LIN {X 0,Y 313.561,Z 316.467,A -85,B 0,C 180,E1 -15772.474,E2 -15772.474} C_VEL
LIN {X 0,Y 320.845,Z 338.006,A -85,B 0,C 180,E1 -15773.542,E2 -15773.542} C_VEL
LIN {X 0,Y 322.386,Z 346.746,A -85,B 0,C 180,E1 -15773.871,E2 -15773.871} C_VEL
LIN {X 0,Y 320.224,Z 424.19,A -85,B 0,C 180,E1 -15775.8,E2 -15775.8} C_VEL
LIN {X 0,Y 319.459,Z 438.164,A -85,B 0,C 180,E1 -15776.412,E2 -15776.412} C_VEL
LIN {X 0,Y 318.685,Z 450.762,A -85,B 0,C 180,E1 -15777.233,E2 -15777.233} C_VEL
LIN {X 0,Y 317.606,Z 462.924,A -85,B 0,C 180,E1 -15778.297,E2 -15778.297} C_VEL
LIN {X 0,Y 316.488,Z 474.165,A -85,B 0,C 180,E1 -15779.558,E2 -15779.558} C_VEL
LIN {X 0,Y 315.388,Z 484.512,A -85,B 0,C 180,E1 -15781.019,E2 -15781.019} C_VEL
LIN {X 0,Y 314.251,Z 493.873,A -85,B 0,C 180,E1 -15782.653,E2 -15782.653} C_VEL
LIN {X 0,Y 313.15,Z 502.541,A -85,B 0,C 180,E1 -15784.52,E2 -15784.52} C_VEL
LIN {X 0,Y 312.337,Z 509.035,A -85,B 0,C 180,E1 -15786.251,E2 -15786.251} C_VEL
LIN {X 0,Y 311.635,Z 515.662,A -85,B 0,C 180,E1 -15788.494,E2 -15788.494} C_VEL
LIN {X 0,Y 311.223,Z 519.919,A -85,B 0,C 180,E1 -15790.35,E2 -15790.35} C_VEL
LIN {X 0,Y 310.751,Z 523.922,A -85,B 0,C 180,E1 -15792.726,E2 -15792.726} C_VEL
LIN {X 0,Y 310.539,Z 525.963,A -85,B 0,C 180,E1 -15794.555,E2 -15794.555} C_VEL
LIN {X 0,Y 310.509,Z 527.474,A -85,B 0,C 180,E1 -15797.233,E2 -15797.233} C_VEL
LIN {X 0,Y 310.562,Z 527.524,A -85,B 0,C 180,E1 -15798.983,E2 -15798.983} C_VEL
LIN {X 0,Y 310.752,Z 526.817,A -85,B 0,C 180,E1 -15800.709,E2 -15800.709} C_VEL
LIN {X 0,Y 311.274,Z 524.504,A -85,B 0,C 180,E1 -15803.25,E2 -15803.25} C_VEL
LIN {X 0,Y 311.79,Z 521.895,A -85,B 0,C 180,E1 -15805.018,E2 -15805.018} C_VEL
LIN {X 0,Y 312.69,Z 517.119,A -85,B 0,C 180,E1 -15807.355,E2 -15807.355} C_VEL
LIN {X 0,Y 313.24,Z 514.23,A -85,B 0,C 180,E1 -15808.473,E2 -15808.473} C_VEL
LIN {X 0,Y 313.144,Z 511.578,A -85,B 0,C 180,E1 -15809.439,E2 -15809.439} C_VEL
LIN {X 0,Y 311.349,Z 506.988,A -85,B 0,C 180,E1 -15811.019,E2 -15811.019} C_VEL
LIN {X 0,Y 309.655,Z 501.778,A -85,B 0,C 180,E1 -15812.544,E2 -15812.544} C_VEL
LIN {X 0,Y 309.708,Z 498.155,A -85,B 0,C 180,E1 -15813.407,E2 -15813.407} C_VEL
LIN {X 0,Y 311.191,Z 489.974,A -85,B 0,C 180,E1 -15815.021,E2 -15815.021} C_VEL
LIN {X 0,Y 312.898,Z 480.264,A -85,B 0,C 180,E1 -15816.569,E2 -15816.569} C_VEL
LIN {X 0,Y 314.489,Z 470.173,A -85,B 0,C 180,E1 -15817.862,E2 -15817.862} C_VEL
LIN {X 0,Y 316.068,Z 458.486,A -85,B 0,C 180,E1 -15819.052,E2 -15819.052} C_VEL
LIN {X 0,Y 317.448,Z 446.076,A -85,B 0,C 180,E1 -15820.015,E2 -15820.015} C_VEL
LIN {X 0,Y 318.404,Z 433.369,A -85,B 0,C 180,E1 -15820.729,E2 -15820.729} C_VEL
LIN {X 0,Y 319.199,Z 419.555,A -85,B 0,C 180,E1 -15821.22,E2 -15821.22} C_VEL
LIN {X 0,Y 321.928,Z 348.78,A -85,B 0,C 180,E1 -15823.058,E2 -15823.058} C_VEL
LIN {X 0,Y 315.974,Z 334.725,A -85,B 0,C 180,E1 -15824.194,E2 -15824.194} C_VEL
LIN {X 0,Y 308.836,Z 320.932,A -85,B 0,C 180,E1 -15825.566,E2 -15825.566} C_VEL
LIN {X 0,Y 307.107,Z 317.583,A -85,B 0,C 180,E1 -15825.927,E2 -15825.927} C_VEL
LIN {X 0,Y 305.593,Z 312.421,A -85,B 0,C 180,E1 -15827.717,E2 -15827.717} C_VEL
LIN {X 0,Y 305.815,Z 312.391,A -85,B 0,C 180,E1 -15832.074,E2 -15832.074} C_VEL
LIN {X 0,Y 305.69,Z 312.409,A -85,B 0,C 180,E1 -15834.723,E2 -15834.723} C_VEL
LIN {X 0,Y 305.958,Z 312.371,A -85,B 0,C 180,E1 -15838.683,E2 -15838.683} C_VEL
LIN {X 0,Y 305.958,Z 312.368,A -85,B 0,C 180,E1 -15841.316,E2 -15841.316} C_VEL
LIN {X 0,Y 305.678,Z 312.408,A -85,B 0,C 180,E1 -15845.276,E2 -15845.276} C_VEL
LIN {X 0,Y 305.767,Z 312.393,A -85,B 0,C 180,E1 -15847.927,E2 -15847.927} C_VEL
LIN {X 0,Y 305.606,Z 312.418,A -85,B 0,C 180,E1 -15851.945,E2 -15851.945} C_VEL
LIN {X 0,Y 305.612,Z 312.417,A -85,B 0,C 180,E1 -15855.015,E2 -15855.015} C_VEL
LIN {X 0,Y 305.544,Z 312.424,A -85,B 0,C 180,E1 -15859.426,E2 -15859.426} C_VEL
LIN {X 0,Y 305.488,Z 312.43,A -85,B 0,C 180,E1 -15863.039,E2 -15863.039} C_VEL
LIN {X 0,Y 305.549,Z 312.423,A -85,B 0,C 180,E1 -15866.226,E2 -15866.226} C_VEL
LIN {X 0,Y 305.49,Z 312.427,A -85,B 0,C 180,E1 -15869.047,E2 -15869.047} C_VEL
LIN {X 0,Y 305.444,Z 312.431,A -85,B 0,C 180,E1 -15871.952,E2 -15871.952} C_VEL
LIN {X 0,Y 305.464,Z 312.43,A -85,B 0,C 180,E1 -15875.113,E2 -15875.113} C_VEL
LIN {X 0,Y 305.442,Z 312.434,A -85,B 0,C 180,E1 -15878.526,E2 -15878.526} C_VEL
LIN {X 0,Y 305.457,Z 312.438,A -85,B 0,C 180,E1 -15882.585,E2 -15882.585} C_VEL
LIN {X 0,Y 305.427,Z 312.438,A -85,B 0,C 180,E1 -15886.345,E2 -15886.345} C_VEL
LIN {X 0,Y 305.46,Z 312.434,A -85,B 0,C 180,E1 -15889.892,E2 -15889.892} C_VEL
LIN {X 0,Y 305.509,Z 312.492,A -85,B 0,C 180,E1 -15894.134,E2 -15894.134} C_VEL
LIN {X 0,Y 308.452,Z 323.369,A -85,B 0,C 180,E1 -15897.885,E2 -15897.885} C_VEL
LIN {X 0,Y 310.938,Z 334.197,A -85,B 0,C 180,E1 -15901.294,E2 -15901.294} C_VEL
LIN {X 0,Y 311.28,Z 335.799,A -85,B 0,C 180,E1 -15901.707,E2 -15901.707} C_VEL
LIN {X 0,Y 314.458,Z 343.704,A -85,B 0,C 180,E1 -15902.366,E2 -15902.366} C_VEL
LIN {X 0,Y 318.425,Z 363.354,A -85,B 0,C 180,E1 -15903.452,E2 -15903.452} C_VEL
LIN {X 0,Y 320.87,Z 381.215,A -85,B 0,C 180,E1 -15904.276,E2 -15904.276} C_VEL
LIN {X 0,Y 318.482,Z 445.12,A -85,B 0,C 180,E1 -15905.948,E2 -15905.948} C_VEL
LIN {X 0,Y 317.369,Z 459.165,A -85,B 0,C 180,E1 -15906.552,E2 -15906.552} C_VEL
LIN {X 0,Y 315.998,Z 471.837,A -85,B 0,C 180,E1 -15907.353,E2 -15907.353} C_VEL
LIN {X 0,Y 314.357,Z 483.549,A -85,B 0,C 180,E1 -15908.352,E2 -15908.352} C_VEL
LIN {X 0,Y 312.61,Z 494.909,A -85,B 0,C 180,E1 -15909.606,E2 -15909.606} C_VEL
LIN {X 0,Y 310.852,Z 505.242,A -85,B 0,C 180,E1 -15911.034,E2 -15911.034} C_VEL
LIN {X 0,Y 309.342,Z 513.737,A -85,B 0,C 180,E1 -15912.48,E2 -15912.48} C_VEL
LIN {X 0,Y 307.656,Z 523.012,A -85,B 0,C 180,E1 -15914.429,E2 -15914.429} C_VEL
LIN {X 0,Y 306.221,Z 530.528,A -85,B 0,C 180,E1 -15916.393,E2 -15916.393} C_VEL
LIN {X 0,Y 305.201,Z 535.652,A -85,B 0,C 180,E1 -15918.038,E2 -15918.038} C_VEL
LIN {X 0,Y 304.451,Z 540.647,A -85,B 0,C 180,E1 -15920.029,E2 -15920.029} C_VEL
LIN {X 0,Y 303.956,Z 544.511,A -85,B 0,C 180,E1 -15922.025,E2 -15922.025} C_VEL
LIN {X 0,Y 303.625,Z 547.846,A -85,B 0,C 180,E1 -15924.455,E2 -15924.455} C_VEL
LIN {X 0,Y 303.631,Z 549.216,A -85,B 0,C 180,E1 -15926.017,E2 -15926.017} C_VEL
LIN {X 0,Y 303.623,Z 549.939,A -85,B 0,C 180,E1 -15927.346,E2 -15927.346} C_VEL
LIN {X 0,Y 303.613,Z 550.264,A -85,B 0,C 180,E1 -15928.673,E2 -15928.673} C_VEL
LIN {X 0,Y 303.669,Z 550.168,A -85,B 0,C 180,E1 -15929.999,E2 -15929.999} C_VEL
LIN {X 0,Y 303.626,Z 549.623,A -85,B 0,C 180,E1 -15931.326,E2 -15931.326} C_VEL
LIN {X 0,Y 303.63,Z 548.674,A -85,B 0,C 180,E1 -15932.653,E2 -15932.653} C_VEL
LIN {X 0,Y 303.655,Z 547.312,A -85,B 0,C 180,E1 -15933.981,E2 -15933.981} C_VEL
LIN {X 0,Y 303.665,Z 544.964,A -85,B 0,C 180,E1 -15935.621,E2 -15935.621} C_VEL
LIN {X 0,Y 303.939,Z 540.379,A -85,B 0,C 180,E1 -15937.974,E2 -15937.974} C_VEL
LIN {X 0,Y 304.443,Z 534.159,A -85,B 0,C 180,E1 -15940.305,E2 -15940.305} C_VEL
LIN {X 0,Y 305.146,Z 527.327,A -85,B 0,C 180,E1 -15942.3,E2 -15942.3} C_VEL
LIN {X 0,Y 306.186,Z 518.829,A -85,B 0,C 180,E1 -15944.284,E2 -15944.284} C_VEL
LIN {X 0,Y 307.231,Z 510.041,A -85,B 0,C 180,E1 -15945.932,E2 -15945.932} C_VEL
LIN {X 0,Y 308.372,Z 500.41,A -85,B 0,C 180,E1 -15947.404,E2 -15947.404} C_VEL
LIN {X 0,Y 309.563,Z 489.924,A -85,B 0,C 180,E1 -15948.703,E2 -15948.703} C_VEL
LIN {X 0,Y 310.837,Z 478.475,A -85,B 0,C 180,E1 -15949.824,E2 -15949.824} C_VEL
LIN {X 0,Y 312.023,Z 465.463,A -85,B 0,C 180,E1 -15950.777,E2 -15950.777} C_VEL
LIN {X 0,Y 312.903,Z 452.597,A -85,B 0,C 180,E1 -15951.449,E2 -15951.449} C_VEL
LIN {X 0,Y 313.47,Z 439.226,A -85,B 0,C 180,E1 -15951.883,E2 -15951.883} C_VEL
LIN {X 0,Y 314.956,Z 378.874,A -85,B 0,C 180,E1 -15953.412,E2 -15953.412} C_VEL
LIN {X 0,Y 309.275,Z 338.42,A -85,B 0,C 180,E1 -15954.905,E2 -15954.905} C_VEL
LIN {X 0,Y 309.725,Z 333.405,A -85,B 0,C 180,E1 -15956.261,E2 -15956.261} C_VEL
LIN {X 0,Y 307.875,Z 323.557,A -85,B 0,C 180,E1 -15959.147,E2 -15959.147} C_VEL
LIN {X 0,Y 305.484,Z 312.437,A -85,B 0,C 180,E1 -15962.58,E2 -15962.58} C_VEL
LIN {X 0,Y 305.472,Z 312.434,A -85,B 0,C 180,E1 -15966.739,E2 -15966.739} C_VEL
LIN {X 0,Y 305.451,Z 312.437,A -85,B 0,C 180,E1 -15970.599,E2 -15970.599} C_VEL
LIN {X 0,Y 305.422,Z 312.437,A -85,B 0,C 180,E1 -15973.654,E2 -15973.654} C_VEL
LIN {X 0,Y 305.451,Z 312.434,A -85,B 0,C 180,E1 -15977.413,E2 -15977.413} C_VEL
LIN {X 0,Y 305.491,Z 312.429,A -85,B 0,C 180,E1 -15981.6,E2 -15981.6} C_VEL
LIN {X 0,Y 305.458,Z 312.437,A -85,B 0,C 180,E1 -15984.886,E2 -15984.886} C_VEL
LIN {X 0,Y 305.444,Z 312.434,A -85,B 0,C 180,E1 -15988.355,E2 -15988.355} C_VEL
LIN {X 0,Y 305.508,Z 312.429,A -85,B 0,C 180,E1 -15991.113,E2 -15991.113} C_VEL
LIN {X 0,Y 305.56,Z 312.42,A -85,B 0,C 180,E1 -15994.087,E2 -15994.087} C_VEL
LIN {X 0,Y 305.495,Z 312.428,A -85,B 0,C 180,E1 -15998.403,E2 -15998.403} C_VEL
LIN {X 0,Y 305.585,Z 312.422,A -85,B 0,C 180,E1 -16001.218,E2 -16001.218} C_VEL
LIN {X 0,Y 305.644,Z 312.414,A -85,B 0,C 180,E1 -16005.349,E2 -16005.349} C_VEL
LIN {X 0,Y 305.633,Z 312.415,A -85,B 0,C 180,E1 -16009.4,E2 -16009.4} C_VEL
LIN {X 0,Y 305.807,Z 312.39,A -85,B 0,C 180,E1 -16012.074,E2 -16012.074} C_VEL
LIN {X 0,Y 305.683,Z 312.404,A -85,B 0,C 180,E1 -16014.724,E2 -16014.724} C_VEL
LIN {X 0,Y 305.951,Z 312.368,A -85,B 0,C 180,E1 -16018.684,E2 -16018.684} C_VEL
LIN {X 0,Y 305.95,Z 312.371,A -85,B 0,C 180,E1 -16021.317,E2 -16021.317} C_VEL
LIN {X 0,Y 305.671,Z 312.406,A -85,B 0,C 180,E1 -16025.277,E2 -16025.277} C_VEL
LIN {X 0,Y 305.76,Z 312.399,A -85,B 0,C 180,E1 -16027.927,E2 -16027.927} C_VEL
LIN {X 0,Y 305.598,Z 312.417,A -85,B 0,C 180,E1 -16031.946,E2 -16031.946} C_VEL
LIN {X 0,Y 305.633,Z 312.409,A -85,B 0,C 180,E1 -16035.035,E2 -16035.035} C_VEL
LIN {X 0,Y 305.575,Z 312.419,A -85,B 0,C 180,E1 -16038.784,E2 -16038.784} C_VEL
LIN {X 0,Y 305.482,Z 312.428,A -85,B 0,C 180,E1 -16043.04,E2 -16043.04} C_VEL
LIN {X 0,Y 305.466,Z 312.431,A -85,B 0,C 180,E1 -16046.198,E2 -16046.198} C_VEL
LIN {X 0,Y 305.454,Z 312.433,A -85,B 0,C 180,E1 -16049.038,E2 -16049.038} C_VEL
LIN {X 0,Y 305.433,Z 312.436,A -85,B 0,C 180,E1 -16051.954,E2 -16051.954} C_VEL
LIN {X 0,Y 305.459,Z 312.434,A -85,B 0,C 180,E1 -16055.114,E2 -16055.114} C_VEL
LIN {X 0,Y 305.432,Z 312.438,A -85,B 0,C 180,E1 -16058.526,E2 -16058.526} C_VEL
LIN {X 0,Y 305.437,Z 312.433,A -85,B 0,C 180,E1 -16061.858,E2 -16061.858} C_VEL
LIN {X 0,Y 305.398,Z 312.441,A -85,B 0,C 180,E1 -16065.512,E2 -16065.512} C_VEL
LIN {X 0,Y 305.41,Z 312.438,A -85,B 0,C 180,E1 -16068.139,E2 -16068.139} C_VEL
LIN {X 0,Y 305.459,Z 312.432,A -85,B 0,C 180,E1 -16071.596,E2 -16071.596} C_VEL
LIN {X 0,Y 305.462,Z 312.433,A -85,B 0,C 180,E1 -16074.888,E2 -16074.888} C_VEL
LIN {X 0,Y 305.442,Z 312.434,A -85,B 0,C 180,E1 -16078.359,E2 -16078.359} C_VEL
LIN {X 0,Y 305.475,Z 312.433,A -85,B 0,C 180,E1 -16081.11,E2 -16081.11} C_VEL
LIN {X 0,Y 305.499,Z 312.428,A -85,B 0,C 180,E1 -16084.082,E2 -16084.082} C_VEL
LIN {X 0,Y 305.475,Z 312.43,A -85,B 0,C 180,E1 -16088.402,E2 -16088.402} C_VEL
LIN {X 0,Y 305.545,Z 312.423,A -85,B 0,C 180,E1 -16091.216,E2 -16091.216} C_VEL
LIN {X 0,Y 305.63,Z 312.413,A -85,B 0,C 180,E1 -16095.349,E2 -16095.349} C_VEL
LIN {X 0,Y 305.626,Z 312.413,A -85,B 0,C 180,E1 -16099.4,E2 -16099.4} C_VEL
LIN {X 0,Y 305.749,Z 312.401,A -85,B 0,C 180,E1 -16102.074,E2 -16102.074} C_VEL
LIN {X 0,Y 305.656,Z 312.409,A -85,B 0,C 180,E1 -16104.724,E2 -16104.724} C_VEL
LIN {X 0,Y 305.934,Z 312.375,A -85,B 0,C 180,E1 -16108.684,E2 -16108.684} C_VEL
LIN {X 0,Y 305.934,Z 312.374,A -85,B 0,C 180,E1 -16111.317,E2 -16111.317} C_VEL
LIN {X 0,Y 305.789,Z 312.395,A -85,B 0,C 180,E1 -16116.599,E2 -16116.599} C_VEL
LIN {X 0,Y 305.687,Z 312.404,A -85,B 0,C 180,E1 -16119.262,E2 -16119.262} C_VEL
LIN {X 0,Y 305.557,Z 312.421,A -85,B 0,C 180,E1 -16123.298,E2 -16123.298} C_VEL
LIN {X 0,Y 305.5,Z 312.429,A -85,B 0,C 180,E1 -16126.026,E2 -16126.026} C_VEL
LIN {X 0,Y 305.507,Z 312.43,A -85,B 0,C 180,E1 -16130.186,E2 -16130.186} C_VEL
LIN {X 0,Y 305.539,Z 312.645,A -85,B 0,C 180,E1 -16130.624,E2 -16130.624} C_VEL
LIN {X 0,Y 306.386,Z 316.706,A -85,B 0,C 180,E1 -16131.974,E2 -16131.974} C_VEL
LIN {X 0,Y 314.265,Z 339.597,A -85,B 0,C 180,E1 -16133.157,E2 -16133.157} C_VEL
LIN {X 0,Y 315.68,Z 347.88,A -85,B 0,C 180,E1 -16133.474,E2 -16133.474} C_VEL
LIN {X 0,Y 313.45,Z 424.389,A -85,B 0,C 180,E1 -16135.424,E2 -16135.424} C_VEL
LIN {X 0,Y 312.68,Z 438.133,A -85,B 0,C 180,E1 -16136.036,E2 -16136.036} C_VEL
LIN {X 0,Y 311.857,Z 450.91,A -85,B 0,C 180,E1 -16136.881,E2 -16136.881} C_VEL
LIN {X 0,Y 310.757,Z 463.159,A -85,B 0,C 180,E1 -16137.975,E2 -16137.975} C_VEL
LIN {X 0,Y 309.631,Z 473.993,A -85,B 0,C 180,E1 -16139.21,E2 -16139.21} C_VEL
LIN {X 0,Y 308.502,Z 484.193,A -85,B 0,C 180,E1 -16140.66,E2 -16140.66} C_VEL
LIN {X 0,Y 307.265,Z 494.192,A -85,B 0,C 180,E1 -16142.437,E2 -16142.437} C_VEL
LIN {X 0,Y 306.173,Z 502.547,A -85,B 0,C 180,E1 -16144.273,E2 -16144.273} C_VEL
LIN {X 0,Y 305.23,Z 509.94,A -85,B 0,C 180,E1 -16146.303,E2 -16146.303} C_VEL
LIN {X 0,Y 304.539,Z 516.295,A -85,B 0,C 180,E1 -16148.543,E2 -16148.543} C_VEL
LIN {X 0,Y 304.131,Z 520.235,A -85,B 0,C 180,E1 -16150.319,E2 -16150.319} C_VEL
LIN {X 0,Y 303.752,Z 523.501,A -85,B 0,C 180,E1 -16152.234,E2 -16152.234} C_VEL
LIN {X 0,Y 303.487,Z 525.806,A -85,B 0,C 180,E1 -16154.119,E2 -16154.119} C_VEL
LIN {X 0,Y 303.406,Z 527.229,A -85,B 0,C 180,E1 -16155.979,E2 -16155.979} C_VEL
LIN {X 0,Y 303.434,Z 527.824,A -85,B 0,C 180,E1 -16157.832,E2 -16157.832} C_VEL
LIN {X 0,Y 303.537,Z 527.598,A -85,B 0,C 180,E1 -16159.825,E2 -16159.825} C_VEL
LIN {X 0,Y 303.865,Z 526.429,A -85,B 0,C 180,E1 -16161.849,E2 -16161.849} C_VEL
LIN {X 0,Y 304.367,Z 524.234,A -85,B 0,C 180,E1 -16163.918,E2 -16163.918} C_VEL
LIN {X 0,Y 305.079,Z 520.889,A -85,B 0,C 180,E1 -16166.03,E2 -16166.03} C_VEL
LIN {X 0,Y 306.023,Z 516.223,A -85,B 0,C 180,E1 -16168.183,E2 -16168.183} C_VEL
LIN {X 0,Y 307.293,Z 510.044,A -85,B 0,C 180,E1 -16170.353,E2 -16170.353} C_VEL
LIN {X 0,Y 308.954,Z 502.039,A -85,B 0,C 180,E1 -16172.519,E2 -16172.519} C_VEL
LIN {X 0,Y 309.708,Z 498.155,A -85,B 0,C 180,E1 -16173.407,E2 -16173.407} C_VEL
LIN {X 0,Y 309.803,Z 494.364,A -85,B 0,C 180,E1 -16174.248,E2 -16174.248} C_VEL
LIN {X 0,Y 308.349,Z 488.096,A -85,B 0,C 180,E1 -16175.651,E2 -16175.651} C_VEL
LIN {X 0,Y 306.955,Z 481.314,A -85,B 0,C 180,E1 -16176.965,E2 -16176.965} C_VEL
LIN {X 0,Y 307.114,Z 476.728,A -85,B 0,C 180,E1 -16177.654,E2 -16177.654} C_VEL
LIN {X 0,Y 308.772,Z 465.962,A -85,B 0,C 180,E1 -16178.941,E2 -16178.941} C_VEL
LIN {X 0,Y 310.429,Z 453.911,A -85,B 0,C 180,E1 -16180.062,E2 -16180.062} C_VEL
LIN {X 0,Y 311.678,Z 441.042,A -85,B 0,C 180,E1 -16180.973,E2 -16180.973} C_VEL
LIN {X 0,Y 312.603,Z 428.721,A -85,B 0,C 180,E1 -16181.571,E2 -16181.571} C_VEL
LIN {X 0,Y 313.553,Z 407.426,A -85,B 0,C 180,E1 -16182.195,E2 -16182.195} C_VEL
LIN {X 0,Y 315.883,Z 351.291,A -85,B 0,C 180,E1 -16183.681,E2 -16183.681} C_VEL
LIN {X 0,Y 314.794,Z 347.909,A -85,B 0,C 180,E1 -16183.918,E2 -16183.918} C_VEL
LIN {X 0,Y 309.105,Z 335.149,A -85,B 0,C 180,E1 -16185.053,E2 -16185.053} C_VEL
LIN {X 0,Y 301.911,Z 321.533,A -85,B 0,C 180,E1 -16186.517,E2 -16186.517} C_VEL
LIN {X 0,Y 299.925,Z 317.942,A -85,B 0,C 180,E1 -16186.965,E2 -16186.965} C_VEL
LIN {X 0,Y 298.568,Z 313.295,A -85,B 0,C 180,E1 -16188.716,E2 -16188.716} C_VEL
LIN {X 0,Y 298.759,Z 313.27,A -85,B 0,C 180,E1 -16191.886,E2 -16191.886} C_VEL
LIN {X 0,Y 298.661,Z 313.285,A -85,B 0,C 180,E1 -16194.599,E2 -16194.599} C_VEL
LIN {X 0,Y 298.924,Z 313.246,A -85,B 0,C 180,E1 -16198.652,E2 -16198.652} C_VEL
LIN {X 0,Y 298.924,Z 313.244,A -85,B 0,C 180,E1 -16201.347,E2 -16201.347} C_VEL
LIN {X 0,Y 298.646,Z 313.284,A -85,B 0,C 180,E1 -16205.401,E2 -16205.401} C_VEL
LIN {X 0,Y 298.715,Z 313.273,A -85,B 0,C 180,E1 -16208.115,E2 -16208.115} C_VEL
LIN {X 0,Y 298.555,Z 313.296,A -85,B 0,C 180,E1 -16212.231,E2 -16212.231} C_VEL
LIN {X 0,Y 298.552,Z 313.296,A -85,B 0,C 180,E1 -16215.169,E2 -16215.169} C_VEL
LIN {X 0,Y 298.505,Z 313.301,A -85,B 0,C 180,E1 -16219.245,E2 -16219.245} C_VEL
LIN {X 0,Y 298.431,Z 313.307,A -85,B 0,C 180,E1 -16223.6,E2 -16223.6} C_VEL
LIN {X 0,Y 298.491,Z 313.303,A -85,B 0,C 180,E1 -16226.574,E2 -16226.574} C_VEL
LIN {X 0,Y 298.419,Z 313.312,A -85,B 0,C 180,E1 -16229.641,E2 -16229.641} C_VEL
LIN {X 0,Y 298.397,Z 313.314,A -85,B 0,C 180,E1 -16232.8,E2 -16232.8} C_VEL
LIN {X 0,Y 298.446,Z 313.31,A -85,B 0,C 180,E1 -16236.807,E2 -16236.807} C_VEL
LIN {X 0,Y 298.389,Z 313.313,A -85,B 0,C 180,E1 -16241.087,E2 -16241.087} C_VEL
LIN {X 0,Y 298.4,Z 313.313,A -85,B 0,C 180,E1 -16243.103,E2 -16243.103} C_VEL
LIN {X 0,Y 298.405,Z 313.316,A -85,B 0,C 180,E1 -16246.92,E2 -16246.92} C_VEL
LIN {X 0,Y 298.401,Z 313.318,A -85,B 0,C 180,E1 -16251.007,E2 -16251.007} C_VEL
LIN {X 0,Y 298.431,Z 313.333,A -85,B 0,C 180,E1 -16253.196,E2 -16253.196} C_VEL
LIN {X 0,Y 301.052,Z 322.826,A -85,B 0,C 180,E1 -16256.655,E2 -16256.655} C_VEL
LIN {X 0,Y 303.317,Z 332.052,A -85,B 0,C 180,E1 -16259.738,E2 -16259.738} C_VEL
LIN {X 0,Y 304.046,Z 335.241,A -85,B 0,C 180,E1 -16260.72,E2 -16260.72} C_VEL
LIN {X 0,Y 308.776,Z 346.249,A -85,B 0,C 180,E1 -16261.73,E2 -16261.73} C_VEL
LIN {X 0,Y 312.278,Z 363.815,A -85,B 0,C 180,E1 -16262.744,E2 -16262.744} C_VEL
LIN {X 0,Y 314.8,Z 381.869,A -85,B 0,C 180,E1 -16263.611,E2 -16263.611} C_VEL
LIN {X 0,Y 312.451,Z 442.334,A -85,B 0,C 180,E1 -16265.232,E2 -16265.232} C_VEL
LIN {X 0,Y 311.479,Z 455.906,A -85,B 0,C 180,E1 -16265.771,E2 -16265.771} C_VEL
LIN {X 0,Y 310.043,Z 468.747,A -85,B 0,C 180,E1 -16266.54,E2 -16266.54} C_VEL
LIN {X 0,Y 308.367,Z 481.179,A -85,B 0,C 180,E1 -16267.557,E2 -16267.557} C_VEL
LIN {X 0,Y 306.945,Z 490.268,A -85,B 0,C 180,E1 -16268.509,E2 -16268.509} C_VEL
LIN {X 0,Y 304.936,Z 501.44,A -85,B 0,C 180,E1 -16269.95,E2 -16269.95} C_VEL
LIN {X 0,Y 303.228,Z 510.515,A -85,B 0,C 180,E1 -16271.416,E2 -16271.416} C_VEL
LIN {X 0,Y 301.444,Z 519.758,A -85,B 0,C 180,E1 -16273.259,E2 -16273.259} C_VEL
LIN {X 0,Y 300.036,Z 527.115,A -85,B 0,C 180,E1 -16275.068,E2 -16275.068} C_VEL
LIN {X 0,Y 298.629,Z 533.778,A -85,B 0,C 180,E1 -16277.08,E2 -16277.08} C_VEL
LIN {X 0,Y 297.682,Z 539.114,A -85,B 0,C 180,E1 -16279.112,E2 -16279.112} C_VEL
LIN {X 0,Y 297.063,Z 543.286,A -85,B 0,C 180,E1 -16281.153,E2 -16281.153} C_VEL
LIN {X 0,Y 296.687,Z 546.397,A -85,B 0,C 180,E1 -16283.197,E2 -16283.197} C_VEL
LIN {X 0,Y 296.552,Z 547.917,A -85,B 0,C 180,E1 -16284.56,E2 -16284.56} C_VEL
LIN {X 0,Y 296.529,Z 549.011,A -85,B 0,C 180,E1 -16285.922,E2 -16285.922} C_VEL
LIN {X 0,Y 296.548,Z 549.709,A -85,B 0,C 180,E1 -16287.282,E2 -16287.282} C_VEL
LIN {X 0,Y 296.53,Z 550.006,A -85,B 0,C 180,E1 -16288.641,E2 -16288.641} C_VEL
LIN {X 0,Y 296.581,Z 549.858,A -85,B 0,C 180,E1 -16289.999,E2 -16289.999} C_VEL
LIN {X 0,Y 296.542,Z 549.288,A -85,B 0,C 180,E1 -16291.357,E2 -16291.357} C_VEL
LIN {X 0,Y 296.555,Z 548.314,A -85,B 0,C 180,E1 -16292.716,E2 -16292.716} C_VEL
LIN {X 0,Y 296.57,Z 546.918,A -85,B 0,C 180,E1 -16294.076,E2 -16294.076} C_VEL
LIN {X 0,Y 296.614,Z 543.94,A -85,B 0,C 180,E1 -16296.119,E2 -16296.119} C_VEL
LIN {X 0,Y 296.873,Z 539.87,A -85,B 0,C 180,E1 -16298.165,E2 -16298.165} C_VEL
LIN {X 0,Y 297.415,Z 533.556,A -85,B 0,C 180,E1 -16300.552,E2 -16300.552} C_VEL
LIN {X 0,Y 298.185,Z 526.648,A -85,B 0,C 180,E1 -16302.592,E2 -16302.592} C_VEL
LIN {X 0,Y 299.061,Z 519.586,A -85,B 0,C 180,E1 -16304.284,E2 -16304.284} C_VEL
LIN {X 0,Y 300.149,Z 511.068,A -85,B 0,C 180,E1 -16305.969,E2 -16305.969} C_VEL
LIN {X 0,Y 301.272,Z 501.84,A -85,B 0,C 180,E1 -16307.46,E2 -16307.46} C_VEL
LIN {X 0,Y 302.493,Z 491.562,A -85,B 0,C 180,E1 -16308.805,E2 -16308.805} C_VEL
LIN {X 0,Y 303.738,Z 480.555,A -85,B 0,C 180,E1 -16309.955,E2 -16309.955} C_VEL
LIN {X 0,Y 304.923,Z 468.474,A -85,B 0,C 180,E1 -16310.93,E2 -16310.93} C_VEL
LIN {X 0,Y 305.909,Z 456.137,A -85,B 0,C 180,E1 -16311.654,E2 -16311.654} C_VEL
LIN {X 0,Y 306.601,Z 442.461,A -85,B 0,C 180,E1 -16312.178,E2 -16312.178} C_VEL
LIN {X 0,Y 308.158,Z 379.055,A -85,B 0,C 180,E1 -16313.838,E2 -16313.838} C_VEL
LIN {X 0,Y 302.458,Z 338.172,A -85,B 0,C 180,E1 -16315.388,E2 -16315.388} C_VEL
LIN {X 0,Y 302.662,Z 334.001,A -85,B 0,C 180,E1 -16316.55,E2 -16316.55} C_VEL
LIN {X 0,Y 300.848,Z 324.6,A -85,B 0,C 180,E1 -16319.377,E2 -16319.377} C_VEL
LIN {X 0,Y 298.449,Z 313.313,A -85,B 0,C 180,E1 -16322.943,E2 -16322.943} C_VEL
LIN {X 0,Y 298.443,Z 313.31,A -85,B 0,C 180,E1 -16326.807,E2 -16326.807} C_VEL
LIN {X 0,Y 298.405,Z 313.312,A -85,B 0,C 180,E1 -16329.485,E2 -16329.485} C_VEL
LIN {X 0,Y 298.395,Z 313.313,A -85,B 0,C 180,E1 -16333.103,E2 -16333.103} C_VEL
LIN {X 0,Y 298.399,Z 313.315,A -85,B 0,C 180,E1 -16336.92,E2 -16336.92} C_VEL
LIN {X 0,Y 298.411,Z 313.313,A -85,B 0,C 180,E1 -16341.003,E2 -16341.003} C_VEL
LIN {X 0,Y 298.428,Z 313.308,A -85,B 0,C 180,E1 -16343.932,E2 -16343.932} C_VEL
LIN {X 0,Y 298.388,Z 313.311,A -85,B 0,C 180,E1 -16347.983,E2 -16347.983} C_VEL
LIN {X 0,Y 298.452,Z 313.304,A -85,B 0,C 180,E1 -16351.903,E2 -16351.903} C_VEL
LIN {X 0,Y 298.478,Z 313.307,A -85,B 0,C 180,E1 -16354.924,E2 -16354.924} C_VEL
LIN {X 0,Y 298.445,Z 313.309,A -85,B 0,C 180,E1 -16359.315,E2 -16359.315} C_VEL
LIN {X 0,Y 298.532,Z 313.295,A -85,B 0,C 180,E1 -16362.179,E2 -16362.179} C_VEL
LIN {X 0,Y 298.588,Z 313.291,A -85,B 0,C 180,E1 -16364.995,E2 -16364.995} C_VEL
LIN {X 0,Y 298.588,Z 313.289,A -85,B 0,C 180,E1 -16369.147,E2 -16369.147} C_VEL
LIN {X 0,Y 298.753,Z 313.27,A -85,B 0,C 180,E1 -16371.886,E2 -16371.886} C_VEL
LIN {X 0,Y 298.654,Z 313.28,A -85,B 0,C 180,E1 -16374.599,E2 -16374.599} C_VEL
LIN {X 0,Y 298.918,Z 313.244,A -85,B 0,C 180,E1 -16378.653,E2 -16378.653} C_VEL
LIN {X 0,Y 298.916,Z 313.247,A -85,B 0,C 180,E1 -16381.348,E2 -16381.348} C_VEL
LIN {X 0,Y 298.639,Z 313.283,A -85,B 0,C 180,E1 -16385.402,E2 -16385.402} C_VEL
LIN {X 0,Y 298.708,Z 313.275,A -85,B 0,C 180,E1 -16388.116,E2 -16388.116} C_VEL
LIN {X 0,Y 298.548,Z 313.294,A -85,B 0,C 180,E1 -16392.232,E2 -16392.232} C_VEL
LIN {X 0,Y 298.601,Z 313.285,A -85,B 0,C 180,E1 -16395.21,E2 -16395.21} C_VEL
LIN {X 0,Y 298.521,Z 313.296,A -85,B 0,C 180,E1 -16399.245,E2 -16399.245} C_VEL
LIN {X 0,Y 298.416,Z 313.307,A -85,B 0,C 180,E1 -16403.602,E2 -16403.602} C_VEL
LIN {X 0,Y 298.405,Z 313.313,A -85,B 0,C 180,E1 -16406.583,E2 -16406.583} C_VEL
LIN {X 0,Y 298.394,Z 313.311,A -85,B 0,C 180,E1 -16409.644,E2 -16409.644} C_VEL
LIN {X 0,Y 298.389,Z 313.317,A -85,B 0,C 180,E1 -16412.802,E2 -16412.802} C_VEL
LIN {X 0,Y 298.439,Z 313.31,A -85,B 0,C 180,E1 -16416.808,E2 -16416.808} C_VEL
LIN {X 0,Y 298.384,Z 313.315,A -85,B 0,C 180,E1 -16421.089,E2 -16421.089} C_VEL
LIN {X 0,Y 298.397,Z 313.315,A -85,B 0,C 180,E1 -16423.104,E2 -16423.104} C_VEL
LIN {X 0,Y 298.37,Z 313.32,A -85,B 0,C 180,E1 -16426.916,E2 -16426.916} C_VEL
LIN {X 0,Y 298.383,Z 313.317,A -85,B 0,C 180,E1 -16431.012,E2 -16431.012} C_VEL
LIN {X 0,Y 298.416,Z 313.308,A -85,B 0,C 180,E1 -16433.931,E2 -16433.931} C_VEL
LIN {X 0,Y 298.393,Z 313.317,A -85,B 0,C 180,E1 -16437.201,E2 -16437.201} C_VEL
LIN {X 0,Y 298.402,Z 313.311,A -85,B 0,C 180,E1 -16440.626,E2 -16440.626} C_VEL
LIN {X 0,Y 298.439,Z 313.308,A -85,B 0,C 180,E1 -16444.921,E2 -16444.921} C_VEL
LIN {X 0,Y 298.409,Z 313.313,A -85,B 0,C 180,E1 -16447.864,E2 -16447.864} C_VEL
LIN {X 0,Y 298.505,Z 313.298,A -85,B 0,C 180,E1 -16450.756,E2 -16450.756} C_VEL
LIN {X 0,Y 298.588,Z 313.288,A -85,B 0,C 180,E1 -16454.995,E2 -16454.995} C_VEL
LIN {X 0,Y 298.585,Z 313.289,A -85,B 0,C 180,E1 -16459.147,E2 -16459.147} C_VEL
LIN {X 0,Y 298.701,Z 313.279,A -85,B 0,C 180,E1 -16461.885,E2 -16461.885} C_VEL
LIN {X 0,Y 298.627,Z 313.285,A -85,B 0,C 180,E1 -16464.599,E2 -16464.599} C_VEL
LIN {X 0,Y 298.902,Z 313.251,A -85,B 0,C 180,E1 -16468.653,E2 -16468.653} C_VEL
LIN {X 0,Y 298.902,Z 313.25,A -85,B 0,C 180,E1 -16471.348,E2 -16471.348} C_VEL
LIN {X 0,Y 298.737,Z 313.272,A -85,B 0,C 180,E1 -16476.756,E2 -16476.756} C_VEL
LIN {X 0,Y 298.619,Z 313.285,A -85,B 0,C 180,E1 -16479.483,E2 -16479.483} C_VEL
LIN {X 0,Y 298.512,Z 313.298,A -85,B 0,C 180,E1 -16483.618,E2 -16483.618} C_VEL
LIN {X 0,Y 298.444,Z 313.311,A -85,B 0,C 180,E1 -16486.415,E2 -16486.415} C_VEL
LIN {X 0,Y 298.48,Z 313.412,A -85,B 0,C 180,E1 -16490.257,E2 -16490.257} C_VEL
LIN {X 0,Y 299.242,Z 317.071,A -85,B 0,C 180,E1 -16491.484,E2 -16491.484} C_VEL
LIN {X 0,Y 307.897,Z 342.205,A -85,B 0,C 180,E1 -16492.809,E2 -16492.809} C_VEL
LIN {X 0,Y 308.935,Z 348.956,A -85,B 0,C 180,E1 -16493.065,E2 -16493.065} C_VEL
LIN {X 0,Y 306.65,Z 425.17,A -85,B 0,C 180,E1 -16495.065,E2 -16495.065} C_VEL
LIN {X 0,Y 305.831,Z 439.04,A -85,B 0,C 180,E1 -16495.706,E2 -16495.706} C_VEL
LIN {X 0,Y 305.034,Z 451.074,A -85,B 0,C 180,E1 -16496.527,E2 -16496.527} C_VEL
LIN {X 0,Y 304.002,Z 462.334,A -85,B 0,C 180,E1 -16497.541,E2 -16497.541} C_VEL
LIN {X 0,Y 302.685,Z 474.546,A -85,B 0,C 180,E1 -16498.952,E2 -16498.952} C_VEL
LIN {X 0,Y 301.534,Z 484.563,A -85,B 0,C 180,E1 -16500.414,E2 -16500.414} C_VEL
LIN {X 0,Y 300.343,Z 494.038,A -85,B 0,C 180,E1 -16502.129,E2 -16502.129} C_VEL
LIN {X 0,Y 299.25,Z 502.039,A -85,B 0,C 180,E1 -16503.903,E2 -16503.903} C_VEL
LIN {X 0,Y 298.393,Z 508.674,A -85,B 0,C 180,E1 -16505.702,E2 -16505.702} C_VEL
LIN {X 0,Y 297.595,Z 515.137,A -85,B 0,C 180,E1 -16507.881,E2 -16507.881} C_VEL
LIN {X 0,Y 297.069,Z 520.395,A -85,B 0,C 180,E1 -16510.223,E2 -16510.223} C_VEL
LIN {X 0,Y 296.557,Z 524.431,A -85,B 0,C 180,E1 -16512.721,E2 -16512.721} C_VEL
LIN {X 0,Y 296.305,Z 527.055,A -85,B 0,C 180,E1 -16515.363,E2 -16515.363} C_VEL
LIN {X 0,Y 296.327,Z 527.998,A -85,B 0,C 180,E1 -16517.327,E2 -16517.327} C_VEL
LIN {X 0,Y 296.423,Z 528.068,A -85,B 0,C 180,E1 -16519.35,E2 -16519.35} C_VEL
LIN {X 0,Y 296.803,Z 526.768,A -85,B 0,C 180,E1 -16522,E2 -16522} C_VEL
LIN {X 0,Y 297.504,Z 523.939,A -85,B 0,C 180,E1 -16524.635,E2 -16524.635} C_VEL
LIN {X 0,Y 298.472,Z 519.517,A -85,B 0,C 180,E1 -16527.209,E2 -16527.209} C_VEL
LIN {X 0,Y 299.718,Z 513.936,A -85,B 0,C 180,E1 -16529.553,E2 -16529.553} C_VEL
LIN {X 0,Y 301.247,Z 506.879,A -85,B 0,C 180,E1 -16531.807,E2 -16531.807} C_VEL
LIN {X 0,Y 303.008,Z 498.673,A -85,B 0,C 180,E1 -16533.852,E2 -16533.852} C_VEL
LIN {X 0,Y 304.536,Z 490.748,A -85,B 0,C 180,E1 -16535.455,E2 -16535.455} C_VEL
LIN {X 0,Y 306.349,Z 481.084,A -85,B 0,C 180,E1 -16537.045,E2 -16537.045} C_VEL
LIN {X 0,Y 307.114,Z 476.728,A -85,B 0,C 180,E1 -16537.654,E2 -16537.654} C_VEL
LIN {X 0,Y 307.311,Z 471.99,A -85,B 0,C 180,E1 -16538.315,E2 -16538.315} C_VEL
LIN {X 0,Y 306.001,Z 464.244,A -85,B 0,C 180,E1 -16539.443,E2 -16539.443} C_VEL
LIN {X 0,Y 304.609,Z 456.171,A -85,B 0,C 180,E1 -16540.48,E2 -16540.48} C_VEL
LIN {X 0,Y 304.609,Z 450.899,A -85,B 0,C 180,E1 -16540.973,E2 -16540.973} C_VEL
LIN {X 0,Y 305.879,Z 437.278,A -85,B 0,C 180,E1 -16541.864,E2 -16541.864} C_VEL
LIN {X 0,Y 306.794,Z 424.257,A -85,B 0,C 180,E1 -16542.416,E2 -16542.416} C_VEL
LIN {X 0,Y 309.864,Z 352.577,A -85,B 0,C 180,E1 -16544.375,E2 -16544.375} C_VEL
LIN {X 0,Y 304.328,Z 339.73,A -85,B 0,C 180,E1 -16545.54,E2 -16545.54} C_VEL
LIN {X 0,Y 297.274,Z 326.151,A -85,B 0,C 180,E1 -16547.043,E2 -16547.043} C_VEL
LIN {X 0,Y 292.79,Z 318.379,A -85,B 0,C 180,E1 -16548.051,E2 -16548.051} C_VEL
LIN {X 0,Y 291.565,Z 314.166,A -85,B 0,C 180,E1 -16549.672,E2 -16549.672} C_VEL
LIN {X 0,Y 291.748,Z 314.144,A -85,B 0,C 180,E1 -16553.082,E2 -16553.082} C_VEL
LIN {X 0,Y 291.891,Z 314.122,A -85,B 0,C 180,E1 -16558.62,E2 -16558.62} C_VEL
LIN {X 0,Y 291.891,Z 314.12,A -85,B 0,C 180,E1 -16561.379,E2 -16561.379} C_VEL
LIN {X 0,Y 291.615,Z 314.161,A -85,B 0,C 180,E1 -16565.532,E2 -16565.532} C_VEL
LIN {X 0,Y 291.676,Z 314.151,A -85,B 0,C 180,E1 -16568.919,E2 -16568.919} C_VEL
LIN {X 0,Y 291.521,Z 314.169,A -85,B 0,C 180,E1 -16572.531,E2 -16572.531} C_VEL
LIN {X 0,Y 291.509,Z 314.173,A -85,B 0,C 180,E1 -16575.379,E2 -16575.379} C_VEL
LIN {X 0,Y 291.426,Z 314.181,A -85,B 0,C 180,E1 -16579.86,E2 -16579.86} C_VEL
LIN {X 0,Y 291.384,Z 314.18,A -85,B 0,C 180,E1 -16584.206,E2 -16584.206} C_VEL
LIN {X 0,Y 291.423,Z 314.176,A -85,B 0,C 180,E1 -16587.271,E2 -16587.271} C_VEL
LIN {X 0,Y 291.336,Z 314.192,A -85,B 0,C 180,E1 -16590.437,E2 -16590.437} C_VEL
LIN {X 0,Y 291.346,Z 314.192,A -85,B 0,C 180,E1 -16593.698,E2 -16593.698} C_VEL
LIN {X 0,Y 291.374,Z 314.186,A -85,B 0,C 180,E1 -16597.253,E2 -16597.253} C_VEL
LIN {X 0,Y 291.334,Z 314.191,A -85,B 0,C 180,E1 -16600.642,E2 -16600.642} C_VEL
LIN {X 0,Y 291.292,Z 314.202,A -85,B 0,C 180,E1 -16604.401,E2 -16604.401} C_VEL
LIN {X 0,Y 291.328,Z 314.194,A -85,B 0,C 180,E1 -16608.404,E2 -16608.404} C_VEL
LIN {X 0,Y 291.394,Z 314.309,A -85,B 0,C 180,E1 -16612.234,E2 -16612.234} C_VEL
LIN {X 0,Y 293.741,Z 322.444,A -85,B 0,C 180,E1 -16615.372,E2 -16615.372} C_VEL
LIN {X 0,Y 296.124,Z 331.839,A -85,B 0,C 180,E1 -16618.693,E2 -16618.693} C_VEL
LIN {X 0,Y 296.833,Z 334.901,A -85,B 0,C 180,E1 -16619.663,E2 -16619.663} C_VEL
LIN {X 0,Y 302.893,Z 348.131,A -85,B 0,C 180,E1 -16621.007,E2 -16621.007} C_VEL
LIN {X 0,Y 305.318,Z 359.316,A -85,B 0,C 180,E1 -16621.715,E2 -16621.715} C_VEL
LIN {X 0,Y 308.016,Z 376.165,A -85,B 0,C 180,E1 -16622.623,E2 -16622.623} C_VEL
LIN {X 0,Y 308.879,Z 383.748,A -85,B 0,C 180,E1 -16622.972,E2 -16622.972} C_VEL
LIN {X 0,Y 306.116,Z 446.014,A -85,B 0,C 180,E1 -16624.684,E2 -16624.684} C_VEL
LIN {X 0,Y 304.916,Z 459.504,A -85,B 0,C 180,E1 -16625.306,E2 -16625.306} C_VEL
LIN {X 0,Y 303.488,Z 471.335,A -85,B 0,C 180,E1 -16626.092,E2 -16626.092} C_VEL
LIN {X 0,Y 301.591,Z 483.757,A -85,B 0,C 180,E1 -16627.206,E2 -16627.206} C_VEL
LIN {X 0,Y 300.171,Z 492.37,A -85,B 0,C 180,E1 -16628.18,E2 -16628.18} C_VEL
LIN {X 0,Y 298.123,Z 503.001,A -85,B 0,C 180,E1 -16629.651,E2 -16629.651} C_VEL
LIN {X 0,Y 296.164,Z 512.682,A -85,B 0,C 180,E1 -16631.315,E2 -16631.315} C_VEL
LIN {X 0,Y 294.542,Z 520.538,A -85,B 0,C 180,E1 -16632.975,E2 -16632.975} C_VEL
LIN {X 0,Y 292.9,Z 528.484,A -85,B 0,C 180,E1 -16635.051,E2 -16635.051} C_VEL
LIN {X 0,Y 291.266,Z 535.733,A -85,B 0,C 180,E1 -16637.457,E2 -16637.457} C_VEL
LIN {X 0,Y 290.427,Z 540.585,A -85,B 0,C 180,E1 -16639.543,E2 -16639.543} C_VEL
LIN {X 0,Y 289.857,Z 544.321,A -85,B 0,C 180,E1 -16641.634,E2 -16641.634} C_VEL
LIN {X 0,Y 289.604,Z 546.263,A -85,B 0,C 180,E1 -16643.03,E2 -16643.03} C_VEL
LIN {X 0,Y 289.475,Z 547.814,A -85,B 0,C 180,E1 -16644.512,E2 -16644.512} C_VEL
LIN {X 0,Y 289.473,Z 549.481,A -85,B 0,C 180,E1 -16647.216,E2 -16647.216} C_VEL
LIN {X 0,Y 289.45,Z 549.737,A -85,B 0,C 180,E1 -16648.608,E2 -16648.608} C_VEL
LIN {X 0,Y 289.496,Z 549.547,A -85,B 0,C 180,E1 -16649.999,E2 -16649.999} C_VEL
LIN {X 0,Y 289.461,Z 548.949,A -85,B 0,C 180,E1 -16651.39,E2 -16651.39} C_VEL
LIN {X 0,Y 289.482,Z 547.946,A -85,B 0,C 180,E1 -16652.782,E2 -16652.782} C_VEL
LIN {X 0,Y 289.489,Z 546.495,A -85,B 0,C 180,E1 -16654.176,E2 -16654.176} C_VEL
LIN {X 0,Y 289.553,Z 543.457,A -85,B 0,C 180,E1 -16656.27,E2 -16656.27} C_VEL
LIN {X 0,Y 289.828,Z 539.314,A -85,B 0,C 180,E1 -16658.365,E2 -16658.365} C_VEL
LIN {X 0,Y 290.396,Z 532.914,A -85,B 0,C 180,E1 -16660.81,E2 -16660.81} C_VEL
LIN {X 0,Y 291.232,Z 525.921,A -85,B 0,C 180,E1 -16662.897,E2 -16662.897} C_VEL
LIN {X 0,Y 292.127,Z 518.757,A -85,B 0,C 180,E1 -16664.631,E2 -16664.631} C_VEL
LIN {X 0,Y 293.324,Z 509.656,A -85,B 0,C 180,E1 -16666.429,E2 -16666.429} C_VEL
LIN {X 0,Y 294.572,Z 499.37,A -85,B 0,C 180,E1 -16668.068,E2 -16668.068} C_VEL
LIN {X 0,Y 295.924,Z 488.787,A -85,B 0,C 180,E1 -16669.419,E2 -16669.419} C_VEL
LIN {X 0,Y 297.226,Z 477.112,A -85,B 0,C 180,E1 -16670.592,E2 -16670.592} C_VEL
LIN {X 0,Y 298.456,Z 463.838,A -85,B 0,C 180,E1 -16671.587,E2 -16671.587} C_VEL
LIN {X 0,Y 299.421,Z 451.499,A -85,B 0,C 180,E1 -16672.239,E2 -16672.239} C_VEL
LIN {X 0,Y 299.966,Z 436.09,A -85,B 0,C 180,E1 -16672.741,E2 -16672.741} C_VEL
LIN {X 0,Y 301.502,Z 380.544,A -85,B 0,C 180,E1 -16674.217,E2 -16674.217} C_VEL
LIN {X 0,Y 295.662,Z 337.854,A -85,B 0,C 180,E1 -16675.9,E2 -16675.9} C_VEL
LIN {X 0,Y 295.569,Z 334.58,A -85,B 0,C 180,E1 -16676.857,E2 -16676.857} C_VEL
LIN {X 0,Y 293.423,Z 323.792,A -85,B 0,C 180,E1 -16680.197,E2 -16680.197} C_VEL
LIN {X 0,Y 291.394,Z 314.19,A -85,B 0,C 180,E1 -16683.368,E2 -16683.368} C_VEL
LIN {X 0,Y 291.378,Z 314.189,A -85,B 0,C 180,E1 -16687.254,E2 -16687.254} C_VEL
LIN {X 0,Y 291.33,Z 314.196,A -85,B 0,C 180,E1 -16690.641,E2 -16690.641} C_VEL
LIN {X 0,Y 291.287,Z 314.203,A -85,B 0,C 180,E1 -16694.401,E2 -16694.401} C_VEL
LIN {X 0,Y 291.323,Z 314.198,A -85,B 0,C 180,E1 -16698.403,E2 -16698.403} C_VEL
LIN {X 0,Y 291.36,Z 314.191,A -85,B 0,C 180,E1 -16701.16,E2 -16701.16} C_VEL
LIN {X 0,Y 291.381,Z 314.191,A -85,B 0,C 180,E1 -16704.629,E2 -16704.629} C_VEL
LIN {X 0,Y 291.365,Z 314.186,A -85,B 0,C 180,E1 -16707.95,E2 -16707.95} C_VEL
LIN {X 0,Y 291.372,Z 314.189,A -85,B 0,C 180,E1 -16711.157,E2 -16711.157} C_VEL
LIN {X 0,Y 291.407,Z 314.183,A -85,B 0,C 180,E1 -16714.271,E2 -16714.271} C_VEL
LIN {X 0,Y 291.376,Z 314.19,A -85,B 0,C 180,E1 -16717.299,E2 -16717.299} C_VEL
LIN {X 0,Y 291.453,Z 314.176,A -85,B 0,C 180,E1 -16720.27,E2 -16720.27} C_VEL
LIN {X 0,Y 291.55,Z 314.166,A -85,B 0,C 180,E1 -16724.624,E2 -16724.624} C_VEL
LIN {X 0,Y 291.532,Z 314.166,A -85,B 0,C 180,E1 -16728.881,E2 -16728.881} C_VEL
LIN {X 0,Y 291.704,Z 314.15,A -85,B 0,C 180,E1 -16731.689,E2 -16731.689} C_VEL
LIN {X 0,Y 291.625,Z 314.155,A -85,B 0,C 180,E1 -16734.469,E2 -16734.469} C_VEL
LIN {X 0,Y 291.884,Z 314.12,A -85,B 0,C 180,E1 -16738.621,E2 -16738.621} C_VEL
LIN {X 0,Y 291.883,Z 314.123,A -85,B 0,C 180,E1 -16741.38,E2 -16741.38} C_VEL
LIN {X 0,Y 291.653,Z 314.15,A -85,B 0,C 180,E1 -16746.538,E2 -16746.538} C_VEL
LIN {X 0,Y 291.567,Z 314.163,A -85,B 0,C 180,E1 -16749.714,E2 -16749.714} C_VEL
LIN {X 0,Y 291.517,Z 314.169,A -85,B 0,C 180,E1 -16753.951,E2 -16753.951} C_VEL
LIN {X 0,Y 291.481,Z 314.173,A -85,B 0,C 180,E1 -16756.819,E2 -16756.819} C_VEL
LIN {X 0,Y 291.446,Z 314.179,A -85,B 0,C 180,E1 -16759.876,E2 -16759.876} C_VEL
LIN {X 0,Y 291.356,Z 314.19,A -85,B 0,C 180,E1 -16764.21,E2 -16764.21} C_VEL
LIN {X 0,Y 291.353,Z 314.187,A -85,B 0,C 180,E1 -16767.279,E2 -16767.279} C_VEL
LIN {X 0,Y 291.317,Z 314.197,A -85,B 0,C 180,E1 -16770.44,E2 -16770.44} C_VEL
LIN {X 0,Y 291.34,Z 314.191,A -85,B 0,C 180,E1 -16773.7,E2 -16773.7} C_VEL
LIN {X 0,Y 291.366,Z 314.187,A -85,B 0,C 180,E1 -16777.253,E2 -16777.253} C_VEL
LIN {X 0,Y 291.329,Z 314.191,A -85,B 0,C 180,E1 -16780.644,E2 -16780.644} C_VEL
LIN {X 0,Y 291.288,Z 314.198,A -85,B 0,C 180,E1 -16784.403,E2 -16784.403} C_VEL
LIN {X 0,Y 291.294,Z 314.198,A -85,B 0,C 180,E1 -16788.412,E2 -16788.412} C_VEL
LIN {X 0,Y 291.334,Z 314.194,A -85,B 0,C 180,E1 -16791.157,E2 -16791.157} C_VEL
LIN {X 0,Y 291.36,Z 314.188,A -85,B 0,C 180,E1 -16794.627,E2 -16794.627} C_VEL
LIN {X 0,Y 291.366,Z 314.189,A -85,B 0,C 180,E1 -16797.951,E2 -16797.951} C_VEL
LIN {X 0,Y 291.344,Z 314.194,A -85,B 0,C 180,E1 -16801.155,E2 -16801.155} C_VEL
LIN {X 0,Y 291.358,Z 314.189,A -85,B 0,C 180,E1 -16804.268,E2 -16804.268} C_VEL
LIN {X 0,Y 291.368,Z 314.191,A -85,B 0,C 180,E1 -16807.299,E2 -16807.299} C_VEL
LIN {X 0,Y 291.441,Z 314.179,A -85,B 0,C 180,E1 -16810.27,E2 -16810.27} C_VEL
LIN {X 0,Y 291.517,Z 314.169,A -85,B 0,C 180,E1 -16814.654,E2 -16814.654} C_VEL
LIN {X 0,Y 291.531,Z 314.167,A -85,B 0,C 180,E1 -16818.881,E2 -16818.881} C_VEL
LIN {X 0,Y 291.655,Z 314.155,A -85,B 0,C 180,E1 -16821.688,E2 -16821.688} C_VEL
LIN {X 0,Y 291.597,Z 314.161,A -85,B 0,C 180,E1 -16824.469,E2 -16824.469} C_VEL
LIN {X 0,Y 291.869,Z 314.127,A -85,B 0,C 180,E1 -16828.621,E2 -16828.621} C_VEL
LIN {X 0,Y 291.869,Z 314.126,A -85,B 0,C 180,E1 -16831.381,E2 -16831.381} C_VEL
LIN {X 0,Y 291.688,Z 314.15,A -85,B 0,C 180,E1 -16836.92,E2 -16836.92} C_VEL
LIN {X 0,Y 291.565,Z 314.164,A -85,B 0,C 180,E1 -16839.715,E2 -16839.715} C_VEL
LIN {X 0,Y 291.475,Z 314.176,A -85,B 0,C 180,E1 -16843.953,E2 -16843.953} C_VEL
LIN {X 0,Y 291.385,Z 314.189,A -85,B 0,C 180,E1 -16848.274,E2 -16848.274} C_VEL
LIN {X 0,Y 291.421,Z 314.249,A -85,B 0,C 180,E1 -16849.898,E2 -16849.898} C_VEL
LIN {X 0,Y 292.012,Z 317.213,A -85,B 0,C 180,E1 -16850.932,E2 -16850.932} C_VEL
LIN {X 0,Y 301.314,Z 343.743,A -85,B 0,C 180,E1 -16852.406,E2 -16852.406} C_VEL
LIN {X 0,Y 302.224,Z 349.14,A -85,B 0,C 180,E1 -16852.622,E2 -16852.622} C_VEL
LIN {X 0,Y 299.876,Z 425.117,A -85,B 0,C 180,E1 -16854.663,E2 -16854.663} C_VEL
LIN {X 0,Y 299.036,Z 438.88,A -85,B 0,C 180,E1 -16855.306,E2 -16855.306} C_VEL
LIN {X 0,Y 298.272,Z 450.768,A -85,B 0,C 180,E1 -16856.125,E2 -16856.125} C_VEL
LIN {X 0,Y 297.052,Z 463.342,A -85,B 0,C 180,E1 -16857.284,E2 -16857.284} C_VEL
LIN {X 0,Y 295.847,Z 474.345,A -85,B 0,C 180,E1 -16858.589,E2 -16858.589} C_VEL
LIN {X 0,Y 294.666,Z 484.309,A -85,B 0,C 180,E1 -16860.058,E2 -16860.058} C_VEL
LIN {X 0,Y 293.42,Z 493.829,A -85,B 0,C 180,E1 -16861.8,E2 -16861.8} C_VEL
LIN {X 0,Y 292.341,Z 501.724,A -85,B 0,C 180,E1 -16863.569,E2 -16863.569} C_VEL
LIN {X 0,Y 291.245,Z 509.739,A -85,B 0,C 180,E1 -16865.794,E2 -16865.794} C_VEL
LIN {X 0,Y 290.466,Z 516.162,A -85,B 0,C 180,E1 -16868.097,E2 -16868.097} C_VEL
LIN {X 0,Y 290.032,Z 520.313,A -85,B 0,C 180,E1 -16869.991,E2 -16869.991} C_VEL
LIN {X 0,Y 289.593,Z 523.698,A -85,B 0,C 180,E1 -16871.989,E2 -16871.989} C_VEL
LIN {X 0,Y 289.385,Z 525.303,A -85,B 0,C 180,E1 -16873.232,E2 -16873.232} C_VEL
LIN {X 0,Y 289.223,Z 527.17,A -85,B 0,C 180,E1 -16875.195,E2 -16875.195} C_VEL
LIN {X 0,Y 289.246,Z 528.167,A -85,B 0,C 180,E1 -16877.129,E2 -16877.129} C_VEL
LIN {X 0,Y 289.321,Z 528.385,A -85,B 0,C 180,E1 -16879.014,E2 -16879.014} C_VEL
LIN {X 0,Y 289.533,Z 527.844,A -85,B 0,C 180,E1 -16880.965,E2 -16880.965} C_VEL
LIN {X 0,Y 289.974,Z 526.316,A -85,B 0,C 180,E1 -16883.113,E2 -16883.113} C_VEL
LIN {X 0,Y 290.632,Z 523.713,A -85,B 0,C 180,E1 -16885.304,E2 -16885.304} C_VEL
LIN {X 0,Y 291.551,Z 519.904,A -85,B 0,C 180,E1 -16887.533,E2 -16887.533} C_VEL
LIN {X 0,Y 292.769,Z 514.714,A -85,B 0,C 180,E1 -16889.791,E2 -16889.791} C_VEL
LIN {X 0,Y 294.349,Z 507.947,A -85,B 0,C 180,E1 -16892.06,E2 -16892.06} C_VEL
LIN {X 0,Y 296.157,Z 500.04,A -85,B 0,C 180,E1 -16894.119,E2 -16894.119} C_VEL
LIN {X 0,Y 297.993,Z 491.091,A -85,B 0,C 180,E1 -16895.994,E2 -16895.994} C_VEL
LIN {X 0,Y 299.918,Z 481.452,A -85,B 0,C 180,E1 -16897.617,E2 -16897.617} C_VEL
LIN {X 0,Y 301.823,Z 470.628,A -85,B 0,C 180,E1 -16899.064,E2 -16899.064} C_VEL
LIN {X 0,Y 303.513,Z 459.362,A -85,B 0,C 180,E1 -16900.258,E2 -16900.258} C_VEL
LIN {X 0,Y 304.609,Z 450.899,A -85,B 0,C 180,E1 -16900.973,E2 -16900.973} C_VEL
LIN {X 0,Y 304.405,Z 447.308,A -85,B 0,C 180,E1 -16901.309,E2 -16901.309} C_VEL
LIN {X 0,Y 300.485,Z 436.19,A -85,B 0,C 180,E1 -16902.562,E2 -16902.562} C_VEL
LIN {X 0,Y 300.212,Z 432.457,A -85,B 0,C 180,E1 -16902.813,E2 -16902.813} C_VEL
LIN {X 0,Y 301.131,Z 418.164,A -85,B 0,C 180,E1 -16903.307,E2 -16903.307} C_VEL
LIN {X 0,Y 304.036,Z 354.736,A -85,B 0,C 180,E1 -16905.068,E2 -16905.068} C_VEL
LIN {X 0,Y 298.485,Z 342.125,A -85,B 0,C 180,E1 -16906.28,E2 -16906.28} C_VEL
LIN {X 0,Y 292.036,Z 329.704,A -85,B 0,C 180,E1 -16907.733,E2 -16907.733} C_VEL
LIN {X 0,Y 286.994,Z 321.368,A -85,B 0,C 180,E1 -16908.899,E2 -16908.899} C_VEL
LIN {X 0,Y 285.624,Z 318.726,A -85,B 0,C 180,E1 -16909.285,E2 -16909.285} C_VEL
LIN {X 0,Y 284.633,Z 315.032,A -85,B 0,C 180,E1 -16910.823,E2 -16910.823} C_VEL
LIN {X 0,Y 284.699,Z 315.023,A -85,B 0,C 180,E1 -16912.91,E2 -16912.91} C_VEL
LIN {X 0,Y 284.857,Z 314.998,A -85,B 0,C 180,E1 -16918.586,E2 -16918.586} C_VEL
LIN {X 0,Y 284.857,Z 314.997,A -85,B 0,C 180,E1 -16921.413,E2 -16921.413} C_VEL
LIN {X 0,Y 284.657,Z 315.019,A -85,B 0,C 180,E1 -16927.091,E2 -16927.091} C_VEL
LIN {X 0,Y 284.52,Z 315.037,A -85,B 0,C 180,E1 -16929.957,E2 -16929.957} C_VEL
LIN {X 0,Y 284.47,Z 315.043,A -85,B 0,C 180,E1 -16934.303,E2 -16934.303} C_VEL
LIN {X 0,Y 284.377,Z 315.062,A -85,B 0,C 180,E1 -16938.74,E2 -16938.74} C_VEL
LIN {X 0,Y 284.317,Z 315.063,A -85,B 0,C 180,E1 -16941.764,E2 -16941.764} C_VEL
LIN {X 0,Y 284.34,Z 315.057,A -85,B 0,C 180,E1 -16944.846,E2 -16944.846} C_VEL
LIN {X 0,Y 284.33,Z 315.057,A -85,B 0,C 180,E1 -16948.011,E2 -16948.011} C_VEL
LIN {X 0,Y 284.295,Z 315.064,A -85,B 0,C 180,E1 -16951.274,E2 -16951.274} C_VEL
LIN {X 0,Y 284.343,Z 315.061,A -85,B 0,C 180,E1 -16955.348,E2 -16955.348} C_VEL
LIN {X 0,Y 284.31,Z 315.064,A -85,B 0,C 180,E1 -16958.169,E2 -16958.169} C_VEL
LIN {X 0,Y 284.271,Z 315.077,A -85,B 0,C 180,E1 -16962.124,E2 -16962.124} C_VEL
LIN {X 0,Y 284.257,Z 315.075,A -85,B 0,C 180,E1 -16966.189,E2 -16966.189} C_VEL
LIN {X 0,Y 284.308,Z 315.069,A -85,B 0,C 180,E1 -16970.024,E2 -16970.024} C_VEL
LIN {X 0,Y 284.356,Z 315.265,A -85,B 0,C 180,E1 -16971.159,E2 -16971.159} C_VEL
LIN {X 0,Y 286.815,Z 323.33,A -85,B 0,C 180,E1 -16974.478,E2 -16974.478} C_VEL
LIN {X 0,Y 289.355,Z 333.52,A -85,B 0,C 180,E1 -16978.222,E2 -16978.222} C_VEL
LIN {X 0,Y 289.629,Z 334.526,A -85,B 0,C 180,E1 -16978.511,E2 -16978.511} C_VEL
LIN {X 0,Y 296.145,Z 348.073,A -85,B 0,C 180,E1 -16980.041,E2 -16980.041} C_VEL
LIN {X 0,Y 297.918,Z 352.547,A -85,B 0,C 180,E1 -16980.46,E2 -16980.46} C_VEL
LIN {X 0,Y 301.379,Z 371.787,A -85,B 0,C 180,E1 -16981.612,E2 -16981.612} C_VEL
LIN {X 0,Y 302.936,Z 384.331,A -85,B 0,C 180,E1 -16982.245,E2 -16982.245} C_VEL
LIN {X 0,Y 300.122,Z 445.095,A -85,B 0,C 180,E1 -16983.955,E2 -16983.955} C_VEL
LIN {X 0,Y 298.867,Z 458.763,A -85,B 0,C 180,E1 -16984.585,E2 -16984.585} C_VEL
LIN {X 0,Y 297.379,Z 470.715,A -85,B 0,C 180,E1 -16985.383,E2 -16985.383} C_VEL
LIN {X 0,Y 295.407,Z 483.218,A -85,B 0,C 180,E1 -16986.515,E2 -16986.515} C_VEL
LIN {X 0,Y 293.871,Z 491.883,A -85,B 0,C 180,E1 -16987.502,E2 -16987.502} C_VEL
LIN {X 0,Y 291.683,Z 502.555,A -85,B 0,C 180,E1 -16988.997,E2 -16988.997} C_VEL
LIN {X 0,Y 289.455,Z 513.11,A -85,B 0,C 180,E1 -16990.865,E2 -16990.865} C_VEL
LIN {X 0,Y 287.424,Z 522.299,A -85,B 0,C 180,E1 -16992.936,E2 -16992.936} C_VEL
LIN {X 0,Y 285.798,Z 529.766,A -85,B 0,C 180,E1 -16995.036,E2 -16995.036} C_VEL
LIN {X 0,Y 284.312,Z 535.802,A -85,B 0,C 180,E1 -16997.145,E2 -16997.145} C_VEL
LIN {X 0,Y 283.437,Z 540.585,A -85,B 0,C 180,E1 -16999.282,E2 -16999.282} C_VEL
LIN {X 0,Y 282.806,Z 544.254,A -85,B 0,C 180,E1 -17001.424,E2 -17001.424} C_VEL
LIN {X 0,Y 282.551,Z 546.136,A -85,B 0,C 180,E1 -17002.855,E2 -17002.855} C_VEL
LIN {X 0,Y 282.338,Z 548.61,A -85,B 0,C 180,E1 -17005.717,E2 -17005.717} C_VEL
LIN {X 0,Y 282.377,Z 549.253,A -85,B 0,C 180,E1 -17007.146,E2 -17007.146} C_VEL
LIN {X 0,Y 282.371,Z 549.455,A -85,B 0,C 180,E1 -17008.573,E2 -17008.573} C_VEL
LIN {X 0,Y 282.413,Z 549.236,A -85,B 0,C 180,E1 -17009.999,E2 -17009.999} C_VEL
LIN {X 0,Y 282.382,Z 548.61,A -85,B 0,C 180,E1 -17011.425,E2 -17011.425} C_VEL
LIN {X 0,Y 282.411,Z 547.578,A -85,B 0,C 180,E1 -17012.852,E2 -17012.852} C_VEL
LIN {X 0,Y 282.416,Z 544.44,A -85,B 0,C 180,E1 -17015.491,E2 -17015.491} C_VEL
LIN {X 0,Y 282.664,Z 540.275,A -85,B 0,C 180,E1 -17017.859,E2 -17017.859} C_VEL
LIN {X 0,Y 283.079,Z 535.263,A -85,B 0,C 180,E1 -17020.007,E2 -17020.007} C_VEL
LIN {X 0,Y 283.747,Z 528.92,A -85,B 0,C 180,E1 -17022.153,E2 -17022.153} C_VEL
LIN {X 0,Y 284.831,Z 520.966,A -85,B 0,C 180,E1 -17024.284,E2 -17024.284} C_VEL
LIN {X 0,Y 286.067,Z 511.707,A -85,B 0,C 180,E1 -17026.267,E2 -17026.267} C_VEL
LIN {X 0,Y 287.363,Z 501.767,A -85,B 0,C 180,E1 -17027.984,E2 -17027.984} C_VEL
LIN {X 0,Y 288.633,Z 491.741,A -85,B 0,C 180,E1 -17029.375,E2 -17029.375} C_VEL
LIN {X 0,Y 289.933,Z 480.891,A -85,B 0,C 180,E1 -17030.577,E2 -17030.577} C_VEL
LIN {X 0,Y 291.296,Z 467.932,A -85,B 0,C 180,E1 -17031.68,E2 -17031.68} C_VEL
LIN {X 0,Y 292.32,Z 455.589,A -85,B 0,C 180,E1 -17032.436,E2 -17032.436} C_VEL
LIN {X 0,Y 293.042,Z 441.948,A -85,B 0,C 180,E1 -17032.983,E2 -17032.983} C_VEL
LIN {X 0,Y 294.7,Z 380.735,A -85,B 0,C 180,E1 -17034.664,E2 -17034.664} C_VEL
LIN {X 0,Y 288.785,Z 337.654,A -85,B 0,C 180,E1 -17036.407,E2 -17036.407} C_VEL
LIN {X 0,Y 287.538,Z 330.08,A -85,B 0,C 180,E1 -17038.762,E2 -17038.762} C_VEL
LIN {X 0,Y 284.775,Z 317.24,A -85,B 0,C 180,E1 -17042.956,E2 -17042.956} C_VEL
LIN {X 0,Y 284.373,Z 315.066,A -85,B 0,C 180,E1 -17043.729,E2 -17043.729} C_VEL
LIN {X 0,Y 284.316,Z 315.073,A -85,B 0,C 180,E1 -17048.167,E2 -17048.167} C_VEL
LIN {X 0,Y 284.266,Z 315.076,A -85,B 0,C 180,E1 -17052.124,E2 -17052.124} C_VEL
LIN {X 0,Y 284.251,Z 315.077,A -85,B 0,C 180,E1 -17056.189,E2 -17056.189} C_VEL
LIN {X 0,Y 284.303,Z 315.069,A -85,B 0,C 180,E1 -17060.023,E2 -17060.023} C_VEL
LIN {X 0,Y 284.346,Z 315.063,A -85,B 0,C 180,E1 -17063.616,E2 -17063.616} C_VEL
LIN {X 0,Y 284.302,Z 315.067,A -85,B 0,C 180,E1 -17067.189,E2 -17067.189} C_VEL
LIN {X 0,Y 284.35,Z 315.055,A -85,B 0,C 180,E1 -17070.375,E2 -17070.375} C_VEL
LIN {X 0,Y 284.369,Z 315.061,A -85,B 0,C 180,E1 -17073.586,E2 -17073.586} C_VEL
LIN {X 0,Y 284.361,Z 315.064,A -85,B 0,C 180,E1 -17076.707,E2 -17076.707} C_VEL
LIN {X 0,Y 284.399,Z 315.061,A -85,B 0,C 180,E1 -17081.262,E2 -17081.262} C_VEL
LIN {X 0,Y 284.487,Z 315.045,A -85,B 0,C 180,E1 -17084.459,E2 -17084.459} C_VEL
LIN {X 0,Y 284.483,Z 315.042,A -85,B 0,C 180,E1 -17088.602,E2 -17088.602} C_VEL
LIN {X 0,Y 284.654,Z 315.029,A -85,B 0,C 180,E1 -17091.481,E2 -17091.481} C_VEL
LIN {X 0,Y 284.596,Z 315.031,A -85,B 0,C 180,E1 -17094.331,E2 -17094.331} C_VEL
LIN {X 0,Y 284.85,Z 314.995,A -85,B 0,C 180,E1 -17098.587,E2 -17098.587} C_VEL
LIN {X 0,Y 284.849,Z 314.999,A -85,B 0,C 180,E1 -17101.414,E2 -17101.414} C_VEL
LIN {X 0,Y 284.649,Z 315.024,A -85,B 0,C 180,E1 -17107.092,E2 -17107.092} C_VEL
LIN {X 0,Y 284.512,Z 315.042,A -85,B 0,C 180,E1 -17109.958,E2 -17109.958} C_VEL
LIN {X 0,Y 284.477,Z 315.048,A -85,B 0,C 180,E1 -17114.303,E2 -17114.303} C_VEL
LIN {X 0,Y 284.419,Z 315.052,A -85,B 0,C 180,E1 -17117.249,E2 -17117.249} C_VEL
LIN {X 0,Y 284.373,Z 315.063,A -85,B 0,C 180,E1 -17120.243,E2 -17120.243} C_VEL
LIN {X 0,Y 284.317,Z 315.063,A -85,B 0,C 180,E1 -17123.854,E2 -17123.854} C_VEL
LIN {X 0,Y 284.283,Z 315.068,A -85,B 0,C 180,E1 -17128.016,E2 -17128.016} C_VEL
LIN {X 0,Y 284.282,Z 315.071,A -85,B 0,C 180,E1 -17131.277,E2 -17131.277} C_VEL
LIN {X 0,Y 284.337,Z 315.063,A -85,B 0,C 180,E1 -17135.349,E2 -17135.349} C_VEL
LIN {X 0,Y 284.303,Z 315.066,A -85,B 0,C 180,E1 -17138.171,E2 -17138.171} C_VEL
LIN {X 0,Y 284.266,Z 315.07,A -85,B 0,C 180,E1 -17142.125,E2 -17142.125} C_VEL
LIN {X 0,Y 284.253,Z 315.074,A -85,B 0,C 180,E1 -17146.19,E2 -17146.19} C_VEL
LIN {X 0,Y 284.282,Z 315.069,A -85,B 0,C 180,E1 -17150.031,E2 -17150.031} C_VEL
LIN {X 0,Y 284.328,Z 315.064,A -85,B 0,C 180,E1 -17153.615,E2 -17153.615} C_VEL
LIN {X 0,Y 284.306,Z 315.072,A -85,B 0,C 180,E1 -17157.191,E2 -17157.191} C_VEL
LIN {X 0,Y 284.337,Z 315.063,A -85,B 0,C 180,E1 -17160.375,E2 -17160.375} C_VEL
LIN {X 0,Y 284.305,Z 315.072,A -85,B 0,C 180,E1 -17163.58,E2 -17163.58} C_VEL
LIN {X 0,Y 284.329,Z 315.065,A -85,B 0,C 180,E1 -17166.705,E2 -17166.705} C_VEL
LIN {X 0,Y 284.378,Z 315.061,A -85,B 0,C 180,E1 -17169.906,E2 -17169.906} C_VEL
LIN {X 0,Y 284.457,Z 315.049,A -85,B 0,C 180,E1 -17174.488,E2 -17174.488} C_VEL
LIN {X 0,Y 284.484,Z 315.046,A -85,B 0,C 180,E1 -17178.602,E2 -17178.602} C_VEL
LIN {X 0,Y 284.612,Z 315.03,A -85,B 0,C 180,E1 -17181.481,E2 -17181.481} C_VEL
LIN {X 0,Y 284.568,Z 315.038,A -85,B 0,C 180,E1 -17184.331,E2 -17184.331} C_VEL
LIN {X 0,Y 284.836,Z 315.004,A -85,B 0,C 180,E1 -17188.587,E2 -17188.587} C_VEL
LIN {X 0,Y 284.836,Z 315.003,A -85,B 0,C 180,E1 -17191.415,E2 -17191.415} C_VEL
LIN {X 0,Y 284.641,Z 315.027,A -85,B 0,C 180,E1 -17197.092,E2 -17197.092} C_VEL
LIN {X 0,Y 284.513,Z 315.044,A -85,B 0,C 180,E1 -17199.958,E2 -17199.958} C_VEL
LIN {X 0,Y 284.409,Z 315.059,A -85,B 0,C 180,E1 -17204.307,E2 -17204.307} C_VEL
LIN {X 0,Y 284.347,Z 315.065,A -85,B 0,C 180,E1 -17207.254,E2 -17207.254} C_VEL
LIN {X 0,Y 284.367,Z 315.145,A -85,B 0,C 180,E1 -17209.545,E2 -17209.545} C_VEL
LIN {X 0,Y 284.866,Z 317.518,A -85,B 0,C 180,E1 -17210.395,E2 -17210.395} C_VEL
LIN {X 0,Y 294.172,Z 343.88,A -85,B 0,C 180,E1 -17211.902,E2 -17211.902} C_VEL
LIN {X 0,Y 295.303,Z 348.432,A -85,B 0,C 180,E1 -17212.117,E2 -17212.117} C_VEL
LIN {X 0,Y 295.506,Z 352.583,A -85,B 0,C 180,E1 -17212.253,E2 -17212.253} C_VEL
LIN {X 0,Y 293.104,Z 425.38,A -85,B 0,C 180,E1 -17214.254,E2 -17214.254} C_VEL
LIN {X 0,Y 292.264,Z 439.159,A -85,B 0,C 180,E1 -17214.915,E2 -17214.915} C_VEL
LIN {X 0,Y 291.488,Z 450.664,A -85,B 0,C 180,E1 -17215.722,E2 -17215.722} C_VEL
LIN {X 0,Y 290.26,Z 463.086,A -85,B 0,C 180,E1 -17216.88,E2 -17216.88} C_VEL
LIN {X 0,Y 288.914,Z 474.971,A -85,B 0,C 180,E1 -17218.318,E2 -17218.318} C_VEL
LIN {X 0,Y 287.694,Z 485.029,A -85,B 0,C 180,E1 -17219.851,E2 -17219.851} C_VEL
LIN {X 0,Y 286.381,Z 494.496,A -85,B 0,C 180,E1 -17221.639,E2 -17221.639} C_VEL
LIN {X 0,Y 285.272,Z 502.326,A -85,B 0,C 180,E1 -17223.45,E2 -17223.45} C_VEL
LIN {X 0,Y 284.327,Z 509.036,A -85,B 0,C 180,E1 -17225.343,E2 -17225.343} C_VEL
LIN {X 0,Y 283.528,Z 515.239,A -85,B 0,C 180,E1 -17227.513,E2 -17227.513} C_VEL
LIN {X 0,Y 283.013,Z 520.051,A -85,B 0,C 180,E1 -17229.662,E2 -17229.662} C_VEL
LIN {X 0,Y 282.447,Z 524.255,A -85,B 0,C 180,E1 -17232.209,E2 -17232.209} C_VEL
LIN {X 0,Y 282.185,Z 526.567,A -85,B 0,C 180,E1 -17234.216,E2 -17234.216} C_VEL
LIN {X 0,Y 282.105,Z 528.037,A -85,B 0,C 180,E1 -17236.259,E2 -17236.259} C_VEL
LIN {X 0,Y 282.173,Z 528.659,A -85,B 0,C 180,E1 -17238.349,E2 -17238.349} C_VEL
LIN {X 0,Y 282.381,Z 528.401,A -85,B 0,C 180,E1 -17240.493,E2 -17240.493} C_VEL
LIN {X 0,Y 282.954,Z 526.591,A -85,B 0,C 180,E1 -17243.407,E2 -17243.407} C_VEL
LIN {X 0,Y 283.859,Z 523.26,A -85,B 0,C 180,E1 -17246.146,E2 -17246.146} C_VEL
LIN {X 0,Y 285.132,Z 518.341,A -85,B 0,C 180,E1 -17248.827,E2 -17248.827} C_VEL
LIN {X 0,Y 286.667,Z 512.206,A -85,B 0,C 180,E1 -17251.261,E2 -17251.261} C_VEL
LIN {X 0,Y 288.209,Z 506.052,A -85,B 0,C 180,E1 -17253.184,E2 -17253.184} C_VEL
LIN {X 0,Y 290.222,Z 497.507,A -85,B 0,C 180,E1 -17255.323,E2 -17255.323} C_VEL
LIN {X 0,Y 292.224,Z 488.259,A -85,B 0,C 180,E1 -17257.155,E2 -17257.155} C_VEL
LIN {X 0,Y 294.383,Z 477.456,A -85,B 0,C 180,E1 -17258.863,E2 -17258.863} C_VEL
LIN {X 0,Y 296.33,Z 466.265,A -85,B 0,C 180,E1 -17260.247,E2 -17260.247} C_VEL
LIN {X 0,Y 298.079,Z 454.485,A -85,B 0,C 180,E1 -17261.38,E2 -17261.38} C_VEL
LIN {X 0,Y 299.411,Z 441.886,A -85,B 0,C 180,E1 -17262.308,E2 -17262.308} C_VEL
LIN {X 0,Y 300.212,Z 432.457,A -85,B 0,C 180,E1 -17262.813,E2 -17262.813} C_VEL
LIN {X 0,Y 300.095,Z 426.771,A -85,B 0,C 180,E1 -17263.122,E2 -17263.122} C_VEL
LIN {X 0,Y 296.193,Z 408.277,A -85,B 0,C 180,E1 -17264.289,E2 -17264.289} C_VEL
LIN {X 0,Y 295.929,Z 402.488,A -85,B 0,C 180,E1 -17264.513,E2 -17264.513} C_VEL
LIN {X 0,Y 298.207,Z 356.884,A -85,B 0,C 180,E1 -17265.796,E2 -17265.796} C_VEL
LIN {X 0,Y 293.015,Z 345.124,A -85,B 0,C 180,E1 -17267,E2 -17267} C_VEL
LIN {X 0,Y 286.54,Z 332.637,A -85,B 0,C 180,E1 -17268.527,E2 -17268.527} C_VEL
LIN {X 0,Y 280.534,Z 322.714,A -85,B 0,C 180,E1 -17270.013,E2 -17270.013} C_VEL
LIN {X 0,Y 278.57,Z 319.244,A -85,B 0,C 180,E1 -17270.556,E2 -17270.556} C_VEL
LIN {X 0,Y 277.634,Z 315.901,A -85,B 0,C 180,E1 -17272.088,E2 -17272.088} C_VEL
LIN {X 0,Y 277.7,Z 315.896,A -85,B 0,C 180,E1 -17277.098,E2 -17277.098} C_VEL
LIN {X 0,Y 277.874,Z 315.871,A -85,B 0,C 180,E1 -17280,E2 -17280} C_VEL
LIN {X 0,Y 277.699,Z 315.893,A -85,B 0,C 180,E1 -17282.901,E2 -17282.901} C_VEL
LIN {X 0,Y 277.614,Z 315.896,A -85,B 0,C 180,E1 -17287.272,E2 -17287.272} C_VEL
LIN {X 0,Y 277.462,Z 315.915,A -85,B 0,C 180,E1 -17290.213,E2 -17290.213} C_VEL
LIN {X 0,Y 277.417,Z 315.925,A -85,B 0,C 180,E1 -17294.675,E2 -17294.675} C_VEL
LIN {X 0,Y 277.327,Z 315.94,A -85,B 0,C 180,E1 -17299.235,E2 -17299.235} C_VEL
LIN {X 0,Y 277.299,Z 315.935,A -85,B 0,C 180,E1 -17303.923,E2 -17303.923} C_VEL
LIN {X 0,Y 277.327,Z 315.931,A -85,B 0,C 180,E1 -17307.504,E2 -17307.504} C_VEL
LIN {X 0,Y 277.274,Z 315.943,A -85,B 0,C 180,E1 -17310.481,E2 -17310.481} C_VEL
LIN {X 0,Y 277.249,Z 315.947,A -85,B 0,C 180,E1 -17313.895,E2 -17313.895} C_VEL
LIN {X 0,Y 277.266,Z 315.942,A -85,B 0,C 180,E1 -17317.469,E2 -17317.469} C_VEL
LIN {X 0,Y 277.211,Z 315.951,A -85,B 0,C 180,E1 -17321.236,E2 -17321.236} C_VEL
LIN {X 0,Y 277.202,Z 315.955,A -85,B 0,C 180,E1 -17325.226,E2 -17325.226} C_VEL
LIN {X 0,Y 277.224,Z 315.953,A -85,B 0,C 180,E1 -17329.512,E2 -17329.512} C_VEL
LIN {X 0,Y 277.312,Z 316.208,A -85,B 0,C 180,E1 -17329.978,E2 -17329.978} C_VEL
LIN {X 0,Y 279.816,Z 324.237,A -85,B 0,C 180,E1 -17333.488,E2 -17333.488} C_VEL
LIN {X 0,Y 282.344,Z 333.942,A -85,B 0,C 180,E1 -17337.231,E2 -17337.231} C_VEL
LIN {X 0,Y 289.551,Z 348.436,A -85,B 0,C 180,E1 -17339.028,E2 -17339.028} C_VEL
LIN {X 0,Y 292.531,Z 355.525,A -85,B 0,C 180,E1 -17339.763,E2 -17339.763} C_VEL
LIN {X 0,Y 295.593,Z 373.146,A -85,B 0,C 180,E1 -17340.861,E2 -17340.861} C_VEL
LIN {X 0,Y 297.065,Z 385.722,A -85,B 0,C 180,E1 -17341.505,E2 -17341.505} C_VEL
LIN {X 0,Y 294.174,Z 444.632,A -85,B 0,C 180,E1 -17343.196,E2 -17343.196} C_VEL
LIN {X 0,Y 292.798,Z 458.972,A -85,B 0,C 180,E1 -17343.876,E2 -17343.876} C_VEL
LIN {X 0,Y 291.295,Z 470.205,A -85,B 0,C 180,E1 -17344.643,E2 -17344.643} C_VEL
LIN {X 0,Y 289.274,Z 482.704,A -85,B 0,C 180,E1 -17345.795,E2 -17345.795} C_VEL
LIN {X 0,Y 287.586,Z 491.4,A -85,B 0,C 180,E1 -17346.792,E2 -17346.792} C_VEL
LIN {X 0,Y 285.098,Z 503.178,A -85,B 0,C 180,E1 -17348.488,E2 -17348.488} C_VEL
LIN {X 0,Y 283.206,Z 511.807,A -85,B 0,C 180,E1 -17350.048,E2 -17350.048} C_VEL
LIN {X 0,Y 281.138,Z 520.55,A -85,B 0,C 180,E1 -17351.981,E2 -17351.981} C_VEL
LIN {X 0,Y 279.209,Z 528.819,A -85,B 0,C 180,E1 -17354.3,E2 -17354.3} C_VEL
LIN {X 0,Y 277.37,Z 535.88,A -85,B 0,C 180,E1 -17356.817,E2 -17356.817} C_VEL
LIN {X 0,Y 276.432,Z 540.572,A -85,B 0,C 180,E1 -17359.007,E2 -17359.007} C_VEL
LIN {X 0,Y 275.771,Z 544.182,A -85,B 0,C 180,E1 -17361.204,E2 -17361.204} C_VEL
LIN {X 0,Y 275.488,Z 546.004,A -85,B 0,C 180,E1 -17362.671,E2 -17362.671} C_VEL
LIN {X 0,Y 275.248,Z 548.418,A -85,B 0,C 180,E1 -17365.606,E2 -17365.606} C_VEL
LIN {X 0,Y 275.283,Z 549.017,A -85,B 0,C 180,E1 -17367.072,E2 -17367.072} C_VEL
LIN {X 0,Y 275.294,Z 549.168,A -85,B 0,C 180,E1 -17368.536,E2 -17368.536} C_VEL
LIN {X 0,Y 275.332,Z 548.918,A -85,B 0,C 180,E1 -17369.999,E2 -17369.999} C_VEL
LIN {X 0,Y 275.306,Z 548.262,A -85,B 0,C 180,E1 -17371.462,E2 -17371.462} C_VEL
LIN {X 0,Y 275.339,Z 547.181,A -85,B 0,C 180,E1 -17372.925,E2 -17372.925} C_VEL
LIN {X 0,Y 275.332,Z 544.25,A -85,B 0,C 180,E1 -17375.439,E2 -17375.439} C_VEL
LIN {X 0,Y 275.591,Z 539.728,A -85,B 0,C 180,E1 -17378.062,E2 -17378.062} C_VEL
LIN {X 0,Y 276.048,Z 534.642,A -85,B 0,C 180,E1 -17380.265,E2 -17380.265} C_VEL
LIN {X 0,Y 276.773,Z 528.207,A -85,B 0,C 180,E1 -17382.464,E2 -17382.464} C_VEL
LIN {X 0,Y 277.871,Z 520.111,A -85,B 0,C 180,E1 -17384.65,E2 -17384.65} C_VEL
LIN {X 0,Y 279.107,Z 511.252,A -85,B 0,C 180,E1 -17386.577,E2 -17386.577} C_VEL
LIN {X 0,Y 280.411,Z 501.749,A -85,B 0,C 180,E1 -17388.257,E2 -17388.257} C_VEL
LIN {X 0,Y 281.715,Z 491.792,A -85,B 0,C 180,E1 -17389.68,E2 -17389.68} C_VEL
LIN {X 0,Y 283.043,Z 481.017,A -85,B 0,C 180,E1 -17390.911,E2 -17390.911} C_VEL
LIN {X 0,Y 284.438,Z 468.173,A -85,B 0,C 180,E1 -17392.039,E2 -17392.039} C_VEL
LIN {X 0,Y 285.551,Z 455.267,A -85,B 0,C 180,E1 -17392.854,E2 -17392.854} C_VEL
LIN {X 0,Y 286.278,Z 441.634,A -85,B 0,C 180,E1 -17393.414,E2 -17393.414} C_VEL
LIN {X 0,Y 288.066,Z 382.002,A -85,B 0,C 180,E1 -17395.09,E2 -17395.09} C_VEL
LIN {X 0,Y 282.14,Z 339.234,A -85,B 0,C 180,E1 -17396.843,E2 -17396.843} C_VEL
LIN {X 0,Y 281.67,Z 337.318,A -85,B 0,C 180,E1 -17396.987,E2 -17396.987} C_VEL
LIN {X 0,Y 279.722,Z 327.523,A -85,B 0,C 180,E1 -17400.164,E2 -17400.164} C_VEL
LIN {X 0,Y 277.329,Z 315.945,A -85,B 0,C 180,E1 -17404.102,E2 -17404.102} C_VEL
LIN {X 0,Y 277.268,Z 315.951,A -85,B 0,C 180,E1 -17408.208,E2 -17408.208} C_VEL
LIN {X 0,Y 277.211,Z 315.955,A -85,B 0,C 180,E1 -17412.674,E2 -17412.674} C_VEL
LIN {X 0,Y 277.205,Z 315.956,A -85,B 0,C 180,E1 -17416.801,E2 -17416.801} C_VEL
LIN {X 0,Y 277.234,Z 315.954,A -85,B 0,C 180,E1 -17420.672,E2 -17420.672} C_VEL
LIN {X 0,Y 277.299,Z 315.942,A -85,B 0,C 180,E1 -17424.344,E2 -17424.344} C_VEL
LIN {X 0,Y 277.239,Z 315.945,A -85,B 0,C 180,E1 -17427.836,E2 -17427.836} C_VEL
LIN {X 0,Y 277.281,Z 315.943,A -85,B 0,C 180,E1 -17431.212,E2 -17431.212} C_VEL
LIN {X 0,Y 277.306,Z 315.941,A -85,B 0,C 180,E1 -17434.479,E2 -17434.479} C_VEL
LIN {X 0,Y 277.28,Z 315.944,A -85,B 0,C 180,E1 -17437.655,E2 -17437.655} C_VEL
LIN {X 0,Y 277.34,Z 315.935,A -85,B 0,C 180,E1 -17440.766,E2 -17440.766} C_VEL
LIN {X 0,Y 277.429,Z 315.928,A -85,B 0,C 180,E1 -17445.326,E2 -17445.326} C_VEL
LIN {X 0,Y 277.501,Z 315.916,A -85,B 0,C 180,E1 -17449.789,E2 -17449.789} C_VEL
LIN {X 0,Y 277.648,Z 315.897,A -85,B 0,C 180,E1 -17452.729,E2 -17452.729} C_VEL
LIN {X 0,Y 277.816,Z 315.871,A -85,B 0,C 180,E1 -17458.551,E2 -17458.551} C_VEL
LIN {X 0,Y 277.815,Z 315.875,A -85,B 0,C 180,E1 -17461.45,E2 -17461.45} C_VEL
LIN {X 0,Y 277.607,Z 315.901,A -85,B 0,C 180,E1 -17467.273,E2 -17467.273} C_VEL
LIN {X 0,Y 277.455,Z 315.918,A -85,B 0,C 180,E1 -17470.214,E2 -17470.214} C_VEL
LIN {X 0,Y 277.43,Z 315.923,A -85,B 0,C 180,E1 -17474.675,E2 -17474.675} C_VEL
LIN {X 0,Y 277.338,Z 315.934,A -85,B 0,C 180,E1 -17479.235,E2 -17479.235} C_VEL
LIN {X 0,Y 277.278,Z 315.94,A -85,B 0,C 180,E1 -17483.926,E2 -17483.926} C_VEL
LIN {X 0,Y 277.268,Z 315.94,A -85,B 0,C 180,E1 -17487.485,E2 -17487.485} C_VEL
LIN {X 0,Y 277.244,Z 315.95,A -85,B 0,C 180,E1 -17490.474,E2 -17490.474} C_VEL
LIN {X 0,Y 277.243,Z 315.948,A -85,B 0,C 180,E1 -17493.897,E2 -17493.897} C_VEL
LIN {X 0,Y 277.26,Z 315.942,A -85,B 0,C 180,E1 -17497.471,E2 -17497.471} C_VEL
LIN {X 0,Y 277.207,Z 315.95,A -85,B 0,C 180,E1 -17501.238,E2 -17501.238} C_VEL
LIN {X 0,Y 277.199,Z 315.956,A -85,B 0,C 180,E1 -17505.228,E2 -17505.228} C_VEL
LIN {X 0,Y 277.196,Z 315.953,A -85,B 0,C 180,E1 -17509.52,E2 -17509.52} C_VEL
LIN {X 0,Y 277.26,Z 315.941,A -85,B 0,C 180,E1 -17512.531,E2 -17512.531} C_VEL
LIN {X 0,Y 277.246,Z 315.946,A -85,B 0,C 180,E1 -17516.106,E2 -17516.106} C_VEL
LIN {X 0,Y 277.262,Z 315.948,A -85,B 0,C 180,E1 -17519.54,E2 -17519.54} C_VEL
LIN {X 0,Y 277.292,Z 315.942,A -85,B 0,C 180,E1 -17522.858,E2 -17522.858} C_VEL
LIN {X 0,Y 277.283,Z 315.943,A -85,B 0,C 180,E1 -17526.076,E2 -17526.076} C_VEL
LIN {X 0,Y 277.326,Z 315.937,A -85,B 0,C 180,E1 -17530.766,E2 -17530.766} C_VEL
LIN {X 0,Y 277.417,Z 315.927,A -85,B 0,C 180,E1 -17535.326,E2 -17535.326} C_VEL
LIN {X 0,Y 277.46,Z 315.925,A -85,B 0,C 180,E1 -17539.788,E2 -17539.788} C_VEL
LIN {X 0,Y 277.603,Z 315.903,A -85,B 0,C 180,E1 -17542.729,E2 -17542.729} C_VEL
LIN {X 0,Y 277.802,Z 315.88,A -85,B 0,C 180,E1 -17548.551,E2 -17548.551} C_VEL
LIN {X 0,Y 277.801,Z 315.879,A -85,B 0,C 180,E1 -17551.45,E2 -17551.45} C_VEL
LIN {X 0,Y 277.597,Z 315.904,A -85,B 0,C 180,E1 -17557.273,E2 -17557.273} C_VEL
LIN {X 0,Y 277.453,Z 315.925,A -85,B 0,C 180,E1 -17560.214,E2 -17560.214} C_VEL
LIN {X 0,Y 277.368,Z 315.937,A -85,B 0,C 180,E1 -17564.678,E2 -17564.678} C_VEL
LIN {X 0,Y 277.321,Z 316.045,A -85,B 0,C 180,E1 -17569.188,E2 -17569.188} C_VEL
LIN {X 0,Y 277.763,Z 318.001,A -85,B 0,C 180,E1 -17569.846,E2 -17569.846} C_VEL
LIN {X 0,Y 287.569,Z 345.56,A -85,B 0,C 180,E1 -17571.471,E2 -17571.471} C_VEL
LIN {X 0,Y 288.852,Z 350.558,A -85,B 0,C 180,E1 -17571.715,E2 -17571.715} C_VEL
LIN {X 0,Y 286.322,Z 425.839,A -85,B 0,C 180,E1 -17573.844,E2 -17573.844} C_VEL
LIN {X 0,Y 285.454,Z 439.79,A -85,B 0,C 180,E1 -17574.536,E2 -17574.536} C_VEL
LIN {X 0,Y 284.565,Z 451.813,A -85,B 0,C 180,E1 -17575.412,E2 -17575.412} C_VEL
LIN {X 0,Y 283.432,Z 463.195,A -85,B 0,C 180,E1 -17576.509,E2 -17576.509} C_VEL
LIN {X 0,Y 282.141,Z 474.254,A -85,B 0,C 180,E1 -17577.864,E2 -17577.864} C_VEL
LIN {X 0,Y 280.808,Z 484.793,A -85,B 0,C 180,E1 -17579.479,E2 -17579.479} C_VEL
LIN {X 0,Y 279.52,Z 494.089,A -85,B 0,C 180,E1 -17581.254,E2 -17581.254} C_VEL
LIN {X 0,Y 278.114,Z 503.519,A -85,B 0,C 180,E1 -17583.496,E2 -17583.496} C_VEL
LIN {X 0,Y 277.04,Z 510.943,A -85,B 0,C 180,E1 -17585.728,E2 -17585.728} C_VEL
LIN {X 0,Y 276.305,Z 516.772,A -85,B 0,C 180,E1 -17587.953,E2 -17587.953} C_VEL
LIN {X 0,Y 275.806,Z 521.257,A -85,B 0,C 180,E1 -17590.141,E2 -17590.141} C_VEL
LIN {X 0,Y 275.335,Z 524.542,A -85,B 0,C 180,E1 -17592.248,E2 -17592.248} C_VEL
LIN {X 0,Y 275.074,Z 526.865,A -85,B 0,C 180,E1 -17594.324,E2 -17594.324} C_VEL
LIN {X 0,Y 275.006,Z 528.301,A -85,B 0,C 180,E1 -17596.369,E2 -17596.369} C_VEL
LIN {X 0,Y 275.079,Z 528.912,A -85,B 0,C 180,E1 -17598.373,E2 -17598.373} C_VEL
LIN {X 0,Y 275.264,Z 528.794,A -85,B 0,C 180,E1 -17600.334,E2 -17600.334} C_VEL
LIN {X 0,Y 275.604,Z 527.979,A -85,B 0,C 180,E1 -17602.264,E2 -17602.264} C_VEL
LIN {X 0,Y 276.202,Z 526.095,A -85,B 0,C 180,E1 -17604.514,E2 -17604.514} C_VEL
LIN {X 0,Y 277.053,Z 523.086,A -85,B 0,C 180,E1 -17606.837,E2 -17606.837} C_VEL
LIN {X 0,Y 278.234,Z 518.824,A -85,B 0,C 180,E1 -17609.185,E2 -17609.185} C_VEL
LIN {X 0,Y 279.783,Z 513.119,A -85,B 0,C 180,E1 -17611.545,E2 -17611.545} C_VEL
LIN {X 0,Y 281.75,Z 505.779,A -85,B 0,C 180,E1 -17613.896,E2 -17613.896} C_VEL
LIN {X 0,Y 283.508,Z 498.668,A -85,B 0,C 180,E1 -17615.715,E2 -17615.715} C_VEL
LIN {X 0,Y 285.579,Z 489.694,A -85,B 0,C 180,E1 -17617.576,E2 -17617.576} C_VEL
LIN {X 0,Y 287.718,Z 479.556,A -85,B 0,C 180,E1 -17619.256,E2 -17619.256} C_VEL
LIN {X 0,Y 289.837,Z 468.4,A -85,B 0,C 180,E1 -17620.732,E2 -17620.732} C_VEL
LIN {X 0,Y 291.766,Z 456.425,A -85,B 0,C 180,E1 -17621.951,E2 -17621.951} C_VEL
LIN {X 0,Y 293.259,Z 444.143,A -85,B 0,C 180,E1 -17622.907,E2 -17622.907} C_VEL
LIN {X 0,Y 294.389,Z 431.58,A -85,B 0,C 180,E1 -17623.608,E2 -17623.608} C_VEL
LIN {X 0,Y 295.354,Z 415.567,A -85,B 0,C 180,E1 -17624.14,E2 -17624.14} C_VEL
LIN {X 0,Y 295.929,Z 402.488,A -85,B 0,C 180,E1 -17624.513,E2 -17624.513} C_VEL
LIN {X 0,Y 295.699,Z 396.712,A -85,B 0,C 180,E1 -17624.746,E2 -17624.746} C_VEL
LIN {X 0,Y 291.971,Z 378.2,A -85,B 0,C 180,E1 -17625.934,E2 -17625.934} C_VEL
LIN {X 0,Y 291.714,Z 372.429,A -85,B 0,C 180,E1 -17626.184,E2 -17626.184} C_VEL
LIN {X 0,Y 292.35,Z 358.79,A -85,B 0,C 180,E1 -17626.594,E2 -17626.594} C_VEL
LIN {X 0,Y 287.617,Z 348.146,A -85,B 0,C 180,E1 -17627.743,E2 -17627.743} C_VEL
LIN {X 0,Y 281.721,Z 336.675,A -85,B 0,C 180,E1 -17629.216,E2 -17629.216} C_VEL
LIN {X 0,Y 275.42,Z 326.206,A -85,B 0,C 180,E1 -17630.862,E2 -17630.862} C_VEL
LIN {X 0,Y 273.275,Z 322.842,A -85,B 0,C 180,E1 -17631.449,E2 -17631.449} C_VEL
LIN {X 0,Y 271.531,Z 319.637,A -85,B 0,C 180,E1 -17632.003,E2 -17632.003} C_VEL
LIN {X 0,Y 270.568,Z 316.78,A -85,B 0,C 180,E1 -17633.474,E2 -17633.474} C_VEL
LIN {X 0,Y 270.789,Z 316.75,A -85,B 0,C 180,E1 -17638.512,E2 -17638.512} C_VEL
LIN {X 0,Y 270.789,Z 316.749,A -85,B 0,C 180,E1 -17641.487,E2 -17641.487} C_VEL
LIN {X 0,Y 270.574,Z 316.774,A -85,B 0,C 180,E1 -17647.462,E2 -17647.462} C_VEL
LIN {X 0,Y 270.415,Z 316.793,A -85,B 0,C 180,E1 -17650.482,E2 -17650.482} C_VEL
LIN {X 0,Y 270.375,Z 316.806,A -85,B 0,C 180,E1 -17655.066,E2 -17655.066} C_VEL
LIN {X 0,Y 270.263,Z 316.817,A -85,B 0,C 180,E1 -17659.758,E2 -17659.758} C_VEL
LIN {X 0,Y 270.24,Z 316.812,A -85,B 0,C 180,E1 -17664.589,E2 -17664.589} C_VEL
LIN {X 0,Y 270.272,Z 316.808,A -85,B 0,C 180,E1 -17667.908,E2 -17667.908} C_VEL
LIN {X 0,Y 270.186,Z 316.82,A -85,B 0,C 180,E1 -17671.348,E2 -17671.348} C_VEL
LIN {X 0,Y 270.203,Z 316.82,A -85,B 0,C 180,E1 -17674.905,E2 -17674.905} C_VEL
LIN {X 0,Y 270.199,Z 316.825,A -85,B 0,C 180,E1 -17678.71,E2 -17678.71} C_VEL
LIN {X 0,Y 270.167,Z 316.829,A -85,B 0,C 180,E1 -17683.248,E2 -17683.248} C_VEL
LIN {X 0,Y 270.173,Z 316.831,A -85,B 0,C 180,E1 -17687.441,E2 -17687.441} C_VEL
LIN {X 0,Y 270.173,Z 316.959,A -85,B 0,C 180,E1 -17688.555,E2 -17688.555} C_VEL
LIN {X 0,Y 272.554,Z 324.404,A -85,B 0,C 180,E1 -17692.06,E2 -17692.06} C_VEL
LIN {X 0,Y 274.517,Z 331.367,A -85,B 0,C 180,E1 -17695.009,E2 -17695.009} C_VEL
LIN {X 0,Y 275.101,Z 333.576,A -85,B 0,C 180,E1 -17695.841,E2 -17695.841} C_VEL
LIN {X 0,Y 280.892,Z 344.639,A -85,B 0,C 180,E1 -17697.407,E2 -17697.407} C_VEL
LIN {X 0,Y 286.106,Z 355.695,A -85,B 0,C 180,E1 -17698.749,E2 -17698.749} C_VEL
LIN {X 0,Y 287.401,Z 359.38,A -85,B 0,C 180,E1 -17699.1,E2 -17699.1} C_VEL
LIN {X 0,Y 290.401,Z 378.208,A -85,B 0,C 180,E1 -17700.279,E2 -17700.279} C_VEL
LIN {X 0,Y 291.263,Z 387.244,A -85,B 0,C 180,E1 -17700.742,E2 -17700.742} C_VEL
LIN {X 0,Y 288.235,Z 445.284,A -85,B 0,C 180,E1 -17702.45,E2 -17702.45} C_VEL
LIN {X 0,Y 286.78,Z 459.332,A -85,B 0,C 180,E1 -17703.138,E2 -17703.138} C_VEL
LIN {X 0,Y 285.006,Z 471.842,A -85,B 0,C 180,E1 -17704.042,E2 -17704.042} C_VEL
LIN {X 0,Y 282.881,Z 483.932,A -85,B 0,C 180,E1 -17705.212,E2 -17705.212} C_VEL
LIN {X 0,Y 281.153,Z 492.342,A -85,B 0,C 180,E1 -17706.229,E2 -17706.229} C_VEL
LIN {X 0,Y 278.801,Z 502.801,A -85,B 0,C 180,E1 -17707.782,E2 -17707.782} C_VEL
LIN {X 0,Y 276.566,Z 512.3,A -85,B 0,C 180,E1 -17709.548,E2 -17709.548} C_VEL
LIN {X 0,Y 274.285,Z 521.3,A -85,B 0,C 180,E1 -17711.639,E2 -17711.639} C_VEL
LIN {X 0,Y 272.384,Z 529.031,A -85,B 0,C 180,E1 -17713.896,E2 -17713.896} C_VEL
LIN {X 0,Y 270.447,Z 535.967,A -85,B 0,C 180,E1 -17716.474,E2 -17716.474} C_VEL
LIN {X 0,Y 269.425,Z 540.574,A -85,B 0,C 180,E1 -17718.717,E2 -17718.717} C_VEL
LIN {X 0,Y 268.726,Z 544.104,A -85,B 0,C 180,E1 -17720.971,E2 -17720.971} C_VEL
LIN {X 0,Y 268.224,Z 547.25,A -85,B 0,C 180,E1 -17723.983,E2 -17723.983} C_VEL
LIN {X 0,Y 268.161,Z 548.227,A -85,B 0,C 180,E1 -17725.49,E2 -17725.49} C_VEL
LIN {X 0,Y 268.193,Z 548.764,A -85,B 0,C 180,E1 -17726.995,E2 -17726.995} C_VEL
LIN {X 0,Y 268.219,Z 548.882,A -85,B 0,C 180,E1 -17728.498,E2 -17728.498} C_VEL
LIN {X 0,Y 268.253,Z 548.6,A -85,B 0,C 180,E1 -17729.999,E2 -17729.999} C_VEL
LIN {X 0,Y 268.231,Z 547.911,A -85,B 0,C 180,E1 -17731.501,E2 -17731.501} C_VEL
LIN {X 0,Y 268.246,Z 546.761,A -85,B 0,C 180,E1 -17733.003,E2 -17733.003} C_VEL
LIN {X 0,Y 268.233,Z 544.088,A -85,B 0,C 180,E1 -17735.352,E2 -17735.352} C_VEL
LIN {X 0,Y 268.434,Z 540.612,A -85,B 0,C 180,E1 -17737.521,E2 -17737.521} C_VEL
LIN {X 0,Y 268.827,Z 535.836,A -85,B 0,C 180,E1 -17739.783,E2 -17739.783} C_VEL
LIN {X 0,Y 269.639,Z 528.606,A -85,B 0,C 180,E1 -17742.416,E2 -17742.416} C_VEL
LIN {X 0,Y 270.777,Z 520.716,A -85,B 0,C 180,E1 -17744.658,E2 -17744.658} C_VEL
LIN {X 0,Y 271.948,Z 512.614,A -85,B 0,C 180,E1 -17746.514,E2 -17746.514} C_VEL
LIN {X 0,Y 273.311,Z 502.715,A -85,B 0,C 180,E1 -17748.36,E2 -17748.36} C_VEL
LIN {X 0,Y 274.595,Z 493.034,A -85,B 0,C 180,E1 -17749.822,E2 -17749.822} C_VEL
LIN {X 0,Y 275.987,Z 482.696,A -85,B 0,C 180,E1 -17751.08,E2 -17751.08} C_VEL
LIN {X 0,Y 277.414,Z 470.434,A -85,B 0,C 180,E1 -17752.235,E2 -17752.235} C_VEL
LIN {X 0,Y 278.566,Z 457.759,A -85,B 0,C 180,E1 -17753.117,E2 -17753.117} C_VEL
LIN {X 0,Y 279.404,Z 444.826,A -85,B 0,C 180,E1 -17753.731,E2 -17753.731} C_VEL
LIN {X 0,Y 281.356,Z 382.921,A -85,B 0,C 180,E1 -17755.53,E2 -17755.53} C_VEL
LIN {X 0,Y 275.715,Z 341.369,A -85,B 0,C 180,E1 -17757.28,E2 -17757.28} C_VEL
LIN {X 0,Y 274.458,Z 337.139,A -85,B 0,C 180,E1 -17757.549,E2 -17757.549} C_VEL
LIN {X 0,Y 272.323,Z 326.625,A -85,B 0,C 180,E1 -17761.073,E2 -17761.073} C_VEL
LIN {X 0,Y 270.256,Z 316.826,A -85,B 0,C 180,E1 -17764.505,E2 -17764.505} C_VEL
LIN {X 0,Y 270.194,Z 316.83,A -85,B 0,C 180,E1 -17768.71,E2 -17768.71} C_VEL
LIN {X 0,Y 270.168,Z 316.833,A -85,B 0,C 180,E1 -17772.557,E2 -17772.557} C_VEL
LIN {X 0,Y 270.161,Z 316.834,A -85,B 0,C 180,E1 -17776.75,E2 -17776.75} C_VEL
LIN {X 0,Y 270.218,Z 316.824,A -85,B 0,C 180,E1 -17781.282,E2 -17781.282} C_VEL
LIN {X 0,Y 270.21,Z 316.826,A -85,B 0,C 180,E1 -17785.096,E2 -17785.096} C_VEL
LIN {X 0,Y 270.195,Z 316.818,A -85,B 0,C 180,E1 -17789.13,E2 -17789.13} C_VEL
LIN {X 0,Y 270.259,Z 316.815,A -85,B 0,C 180,E1 -17792.146,E2 -17792.146} C_VEL
LIN {X 0,Y 270.272,Z 316.818,A -85,B 0,C 180,E1 -17795.519,E2 -17795.519} C_VEL
LIN {X 0,Y 270.297,Z 316.811,A -85,B 0,C 180,E1 -17800.244,E2 -17800.244} C_VEL
LIN {X 0,Y 270.398,Z 316.802,A -85,B 0,C 180,E1 -17804.935,E2 -17804.935} C_VEL
LIN {X 0,Y 270.436,Z 316.797,A -85,B 0,C 180,E1 -17809.519,E2 -17809.519} C_VEL
LIN {X 0,Y 270.606,Z 316.774,A -85,B 0,C 180,E1 -17812.539,E2 -17812.539} C_VEL
LIN {X 0,Y 270.782,Z 316.746,A -85,B 0,C 180,E1 -17818.513,E2 -17818.513} C_VEL
LIN {X 0,Y 270.781,Z 316.751,A -85,B 0,C 180,E1 -17821.488,E2 -17821.488} C_VEL
LIN {X 0,Y 270.566,Z 316.779,A -85,B 0,C 180,E1 -17827.463,E2 -17827.463} C_VEL
LIN {X 0,Y 270.407,Z 316.793,A -85,B 0,C 180,E1 -17830.483,E2 -17830.483} C_VEL
LIN {X 0,Y 270.398,Z 316.797,A -85,B 0,C 180,E1 -17835.065,E2 -17835.065} C_VEL
LIN {X 0,Y 270.296,Z 316.813,A -85,B 0,C 180,E1 -17839.756,E2 -17839.756} C_VEL
LIN {X 0,Y 270.22,Z 316.816,A -85,B 0,C 180,E1 -17844.591,E2 -17844.591} C_VEL
LIN {X 0,Y 270.198,Z 316.821,A -85,B 0,C 180,E1 -17847.917,E2 -17847.917} C_VEL
LIN {X 0,Y 270.17,Z 316.828,A -85,B 0,C 180,E1 -17851.351,E2 -17851.351} C_VEL
LIN {X 0,Y 270.198,Z 316.827,A -85,B 0,C 180,E1 -17854.907,E2 -17854.907} C_VEL
LIN {X 0,Y 270.195,Z 316.824,A -85,B 0,C 180,E1 -17858.712,E2 -17858.712} C_VEL
LIN {X 0,Y 270.163,Z 316.83,A -85,B 0,C 180,E1 -17863.25,E2 -17863.25} C_VEL
LIN {X 0,Y 270.153,Z 316.832,A -85,B 0,C 180,E1 -17867.44,E2 -17867.44} C_VEL
LIN {X 0,Y 270.206,Z 316.822,A -85,B 0,C 180,E1 -17871.375,E2 -17871.375} C_VEL
LIN {X 0,Y 270.201,Z 316.826,A -85,B 0,C 180,E1 -17875.096,E2 -17875.096} C_VEL
LIN {X 0,Y 270.184,Z 316.83,A -85,B 0,C 180,E1 -17879.138,E2 -17879.138} C_VEL
LIN {X 0,Y 270.223,Z 316.822,A -85,B 0,C 180,E1 -17882.164,E2 -17882.164} C_VEL
LIN {X 0,Y 270.228,Z 316.825,A -85,B 0,C 180,E1 -17885.544,E2 -17885.544} C_VEL
LIN {X 0,Y 270.263,Z 316.817,A -85,B 0,C 180,E1 -17890.243,E2 -17890.243} C_VEL
LIN {X 0,Y 270.376,Z 316.803,A -85,B 0,C 180,E1 -17894.935,E2 -17894.935} C_VEL
LIN {X 0,Y 270.413,Z 316.8,A -85,B 0,C 180,E1 -17899.519,E2 -17899.519} C_VEL
LIN {X 0,Y 270.565,Z 316.781,A -85,B 0,C 180,E1 -17902.538,E2 -17902.538} C_VEL
LIN {X 0,Y 270.765,Z 316.757,A -85,B 0,C 180,E1 -17908.514,E2 -17908.514} C_VEL
LIN {X 0,Y 270.765,Z 316.756,A -85,B 0,C 180,E1 -17911.488,E2 -17911.488} C_VEL
LIN {X 0,Y 270.557,Z 316.781,A -85,B 0,C 180,E1 -17917.463,E2 -17917.463} C_VEL
LIN {X 0,Y 270.385,Z 316.807,A -85,B 0,C 180,E1 -17920.484,E2 -17920.484} C_VEL
LIN {X 0,Y 270.339,Z 316.811,A -85,B 0,C 180,E1 -17925.069,E2 -17925.069} C_VEL
LIN {X 0,Y 270.256,Z 316.827,A -85,B 0,C 180,E1 -17928.773,E2 -17928.773} C_VEL
LIN {X 0,Y 270.546,Z 318.148,A -85,B 0,C 180,E1 -17929.244,E2 -17929.244} C_VEL
LIN {X 0,Y 279.869,Z 343.952,A -85,B 0,C 180,E1 -17930.841,E2 -17930.841} C_VEL
LIN {X 0,Y 282.147,Z 351.47,A -85,B 0,C 180,E1 -17931.25,E2 -17931.25} C_VEL
LIN {X 0,Y 279.547,Z 426.259,A -85,B 0,C 180,E1 -17933.423,E2 -17933.423} C_VEL
LIN {X 0,Y 278.654,Z 440.087,A -85,B 0,C 180,E1 -17934.126,E2 -17934.126} C_VEL
LIN {X 0,Y 277.776,Z 451.819,A -85,B 0,C 180,E1 -17934.999,E2 -17934.999} C_VEL
LIN {X 0,Y 276.515,Z 464.013,A -85,B 0,C 180,E1 -17936.207,E2 -17936.207} C_VEL
LIN {X 0,Y 275.214,Z 474.805,A -85,B 0,C 180,E1 -17937.572,E2 -17937.572} C_VEL
LIN {X 0,Y 273.828,Z 485.326,A -85,B 0,C 180,E1 -17939.232,E2 -17939.232} C_VEL
LIN {X 0,Y 272.508,Z 494.573,A -85,B 0,C 180,E1 -17941.052,E2 -17941.052} C_VEL
LIN {X 0,Y 271.272,Z 502.518,A -85,B 0,C 180,E1 -17942.961,E2 -17942.961} C_VEL
LIN {X 0,Y 270.32,Z 509.098,A -85,B 0,C 180,E1 -17944.889,E2 -17944.889} C_VEL
LIN {X 0,Y 269.512,Z 514.607,A -85,B 0,C 180,E1 -17946.854,E2 -17946.854} C_VEL
LIN {X 0,Y 269,Z 519.114,A -85,B 0,C 180,E1 -17948.832,E2 -17948.832} C_VEL
LIN {X 0,Y 268.547,Z 522.802,A -85,B 0,C 180,E1 -17950.865,E2 -17950.865} C_VEL
LIN {X 0,Y 268.12,Z 525.671,A -85,B 0,C 180,E1 -17952.963,E2 -17952.963} C_VEL
LIN {X 0,Y 267.933,Z 527.684,A -85,B 0,C 180,E1 -17955.091,E2 -17955.091} C_VEL
LIN {X 0,Y 267.926,Z 528.878,A -85,B 0,C 180,E1 -17957.263,E2 -17957.263} C_VEL
LIN {X 0,Y 268.076,Z 529.223,A -85,B 0,C 180,E1 -17959.49,E2 -17959.49} C_VEL
LIN {X 0,Y 268.388,Z 528.655,A -85,B 0,C 180,E1 -17961.775,E2 -17961.775} C_VEL
LIN {X 0,Y 268.984,Z 527.109,A -85,B 0,C 180,E1 -17964.094,E2 -17964.094} C_VEL
LIN {X 0,Y 269.984,Z 523.926,A -85,B 0,C 180,E1 -17966.862,E2 -17966.862} C_VEL
LIN {X 0,Y 271.464,Z 518.955,A -85,B 0,C 180,E1 -17969.734,E2 -17969.734} C_VEL
LIN {X 0,Y 273.353,Z 512.435,A -85,B 0,C 180,E1 -17972.432,E2 -17972.432} C_VEL
LIN {X 0,Y 275.354,Z 505.335,A -85,B 0,C 180,E1 -17974.689,E2 -17974.689} C_VEL
LIN {X 0,Y 277.638,Z 496.507,A -85,B 0,C 180,E1 -17976.898,E2 -17976.898} C_VEL
LIN {X 0,Y 279.938,Z 486.94,A -85,B 0,C 180,E1 -17978.806,E2 -17978.806} C_VEL
LIN {X 0,Y 282.219,Z 476.481,A -85,B 0,C 180,E1 -17980.451,E2 -17980.451} C_VEL
LIN {X 0,Y 284.299,Z 465.551,A -85,B 0,C 180,E1 -17981.814,E2 -17981.814} C_VEL
LIN {X 0,Y 286.248,Z 453.475,A -85,B 0,C 180,E1 -17982.984,E2 -17982.984} C_VEL
LIN {X 0,Y 287.717,Z 440.08,A -85,B 0,C 180,E1 -17983.953,E2 -17983.953} C_VEL
LIN {X 0,Y 288.831,Z 428.322,A -85,B 0,C 180,E1 -17984.52,E2 -17984.52} C_VEL
LIN {X 0,Y 291.714,Z 372.429,A -85,B 0,C 180,E1 -17986.184,E2 -17986.184} C_VEL
LIN {X 0,Y 291.487,Z 368.633,A -85,B 0,C 180,E1 -17986.36,E2 -17986.36} C_VEL
LIN {X 0,Y 289.969,Z 363.358,A -85,B 0,C 180,E1 -17986.792,E2 -17986.792} C_VEL
LIN {X 0,Y 287.581,Z 358.648,A -85,B 0,C 180,E1 -17987.349,E2 -17987.349} C_VEL
LIN {X 0,Y 280.053,Z 346.547,A -85,B 0,C 180,E1 -17989.113,E2 -17989.113} C_VEL
LIN {X 0,Y 274.538,Z 336.519,A -85,B 0,C 180,E1 -17990.584,E2 -17990.584} C_VEL
LIN {X 0,Y 268.974,Z 327.452,A -85,B 0,C 180,E1 -17992.162,E2 -17992.162} C_VEL
LIN {X 0,Y 267.112,Z 324.434,A -85,B 0,C 180,E1 -17992.725,E2 -17992.725} C_VEL
LIN {X 0,Y 264.333,Z 320.155,A -85,B 0,C 180,E1 -17993.607,E2 -17993.607} C_VEL
LIN {X 0,Y 263.424,Z 317.673,A -85,B 0,C 180,E1 -17995.025,E2 -17995.025} C_VEL
LIN {X 0,Y 263.753,Z 317.627,A -85,B 0,C 180,E1 -17998.473,E2 -17998.473} C_VEL
LIN {X 0,Y 263.753,Z 317.626,A -85,B 0,C 180,E1 -18001.527,E2 -18001.527} C_VEL
LIN {X 0,Y 263.536,Z 317.651,A -85,B 0,C 180,E1 -18007.662,E2 -18007.662} C_VEL
LIN {X 0,Y 263.357,Z 317.673,A -85,B 0,C 180,E1 -18010.766,E2 -18010.766} C_VEL
LIN {X 0,Y 263.317,Z 317.686,A -85,B 0,C 180,E1 -18015.48,E2 -18015.48} C_VEL
LIN {X 0,Y 263.241,Z 317.687,A -85,B 0,C 180,E1 -18020.308,E2 -18020.308} C_VEL
LIN {X 0,Y 263.195,Z 317.692,A -85,B 0,C 180,E1 -18025.292,E2 -18025.292} C_VEL
LIN {X 0,Y 263.177,Z 317.694,A -85,B 0,C 180,E1 -18028.73,E2 -18028.73} C_VEL
LIN {X 0,Y 263.135,Z 317.702,A -85,B 0,C 180,E1 -18032.288,E2 -18032.288} C_VEL
LIN {X 0,Y 263.183,Z 317.701,A -85,B 0,C 180,E1 -18036.762,E2 -18036.762} C_VEL
LIN {X 0,Y 263.126,Z 317.707,A -85,B 0,C 180,E1 -18041.593,E2 -18041.593} C_VEL
LIN {X 0,Y 263.107,Z 317.709,A -85,B 0,C 180,E1 -18046.155,E2 -18046.155} C_VEL
LIN {X 0,Y 263.145,Z 317.835,A -85,B 0,C 180,E1 -18047.048,E2 -18047.048} C_VEL
LIN {X 0,Y 265.839,Z 326.155,A -85,B 0,C 180,E1 -18051.249,E2 -18051.249} C_VEL
LIN {X 0,Y 267.866,Z 333.131,A -85,B 0,C 180,E1 -18054.299,E2 -18054.299} C_VEL
LIN {X 0,Y 270.609,Z 338.027,A -85,B 0,C 180,E1 -18055.122,E2 -18055.122} C_VEL
LIN {X 0,Y 276.187,Z 348.725,A -85,B 0,C 180,E1 -18056.708,E2 -18056.708} C_VEL
LIN {X 0,Y 281.468,Z 360.234,A -85,B 0,C 180,E1 -18058.145,E2 -18058.145} C_VEL
LIN {X 0,Y 282.409,Z 363.843,A -85,B 0,C 180,E1 -18058.454,E2 -18058.454} C_VEL
LIN {X 0,Y 284.891,Z 380.659,A -85,B 0,C 180,E1 -18059.512,E2 -18059.512} C_VEL
LIN {X 0,Y 285.581,Z 388.036,A -85,B 0,C 180,E1 -18059.901,E2 -18059.901} C_VEL
LIN {X 0,Y 282.452,Z 444.579,A -85,B 0,C 180,E1 -18061.605,E2 -18061.605} C_VEL
LIN {X 0,Y 281.032,Z 458.329,A -85,B 0,C 180,E1 -18062.29,E2 -18062.29} C_VEL
LIN {X 0,Y 279.343,Z 469.527,A -85,B 0,C 180,E1 -18063.072,E2 -18063.072} C_VEL
LIN {X 0,Y 277.144,Z 482.052,A -85,B 0,C 180,E1 -18064.261,E2 -18064.261} C_VEL
LIN {X 0,Y 274.935,Z 492.039,A -85,B 0,C 180,E1 -18065.455,E2 -18065.455} C_VEL
LIN {X 0,Y 272.582,Z 502.493,A -85,B 0,C 180,E1 -18067.047,E2 -18067.047} C_VEL
LIN {X 0,Y 270.428,Z 511.112,A -85,B 0,C 180,E1 -18068.663,E2 -18068.663} C_VEL
LIN {X 0,Y 267.913,Z 520.334,A -85,B 0,C 180,E1 -18070.798,E2 -18070.798} C_VEL
LIN {X 0,Y 265.867,Z 528.123,A -85,B 0,C 180,E1 -18073.095,E2 -18073.095} C_VEL
LIN {X 0,Y 264.097,Z 534.277,A -85,B 0,C 180,E1 -18075.355,E2 -18075.355} C_VEL
LIN {X 0,Y 262.744,Z 539.193,A -85,B 0,C 180,E1 -18077.643,E2 -18077.643} C_VEL
LIN {X 0,Y 261.922,Z 542.99,A -85,B 0,C 180,E1 -18079.955,E2 -18079.955} C_VEL
LIN {X 0,Y 261.348,Z 545.77,A -85,B 0,C 180,E1 -18082.272,E2 -18082.272} C_VEL
LIN {X 0,Y 261.085,Z 547.754,A -85,B 0,C 180,E1 -18084.862,E2 -18084.862} C_VEL
LIN {X 0,Y 261.105,Z 548.51,A -85,B 0,C 180,E1 -18086.913,E2 -18086.913} C_VEL
LIN {X 0,Y 261.144,Z 548.596,A -85,B 0,C 180,E1 -18088.457,E2 -18088.457} C_VEL
LIN {X 0,Y 261.176,Z 548.282,A -85,B 0,C 180,E1 -18089.999,E2 -18089.999} C_VEL
LIN {X 0,Y 261.158,Z 547.544,A -85,B 0,C 180,E1 -18091.541,E2 -18091.541} C_VEL
LIN {X 0,Y 261.156,Z 546.341,A -85,B 0,C 180,E1 -18093.084,E2 -18093.084} C_VEL
LIN {X 0,Y 261.156,Z 543.862,A -85,B 0,C 180,E1 -18095.307,E2 -18095.307} C_VEL
LIN {X 0,Y 261.359,Z 540.04,A -85,B 0,C 180,E1 -18097.726,E2 -18097.726} C_VEL
LIN {X 0,Y 261.78,Z 535.177,A -85,B 0,C 180,E1 -18100.049,E2 -18100.049} C_VEL
LIN {X 0,Y 262.478,Z 528.993,A -85,B 0,C 180,E1 -18102.368,E2 -18102.368} C_VEL
LIN {X 0,Y 263.664,Z 521.29,A -85,B 0,C 180,E1 -18104.667,E2 -18104.667} C_VEL
LIN {X 0,Y 264.867,Z 513.382,A -85,B 0,C 180,E1 -18106.572,E2 -18106.572} C_VEL
LIN {X 0,Y 266.211,Z 503.681,A -85,B 0,C 180,E1 -18108.468,E2 -18108.468} C_VEL
LIN {X 0,Y 267.69,Z 492.941,A -85,B 0,C 180,E1 -18110.156,E2 -18110.156} C_VEL
LIN {X 0,Y 269.115,Z 482.637,A -85,B 0,C 180,E1 -18111.444,E2 -18111.444} C_VEL
LIN {X 0,Y 270.568,Z 470.453,A -85,B 0,C 180,E1 -18112.627,E2 -18112.627} C_VEL
LIN {X 0,Y 271.823,Z 457.149,A -85,B 0,C 180,E1 -18113.574,E2 -18113.574} C_VEL
LIN {X 0,Y 272.705,Z 443.965,A -85,B 0,C 180,E1 -18114.199,E2 -18114.199} C_VEL
LIN {X 0,Y 274.655,Z 383.54,A -85,B 0,C 180,E1 -18116,E2 -18116} C_VEL
LIN {X 0,Y 269.149,Z 342.869,A -85,B 0,C 180,E1 -18117.769,E2 -18117.769} C_VEL
LIN {X 0,Y 267.192,Z 336.88,A -85,B 0,C 180,E1 -18118.166,E2 -18118.166} C_VEL
LIN {X 0,Y 264.841,Z 325.665,A -85,B 0,C 180,E1 -18122.054,E2 -18122.054} C_VEL
LIN {X 0,Y 263.195,Z 317.704,A -85,B 0,C 180,E1 -18124.976,E2 -18124.976} C_VEL
LIN {X 0,Y 263.159,Z 317.708,A -85,B 0,C 180,E1 -18127.896,E2 -18127.896} C_VEL
LIN {X 0,Y 263.12,Z 317.709,A -85,B 0,C 180,E1 -18131.893,E2 -18131.893} C_VEL
LIN {X 0,Y 263.101,Z 317.712,A -85,B 0,C 180,E1 -18136.154,E2 -18136.154} C_VEL
LIN {X 0,Y 263.111,Z 317.71,A -85,B 0,C 180,E1 -18140.129,E2 -18140.129} C_VEL
LIN {X 0,Y 263.183,Z 317.699,A -85,B 0,C 180,E1 -18144.022,E2 -18144.022} C_VEL
LIN {X 0,Y 263.128,Z 317.702,A -85,B 0,C 180,E1 -18147.711,E2 -18147.711} C_VEL
LIN {X 0,Y 263.195,Z 317.695,A -85,B 0,C 180,E1 -18151.783,E2 -18151.783} C_VEL
LIN {X 0,Y 263.221,Z 317.699,A -85,B 0,C 180,E1 -18155.2,E2 -18155.2} C_VEL
LIN {X 0,Y 263.259,Z 317.688,A -85,B 0,C 180,E1 -18159.693,E2 -18159.693} C_VEL
LIN {X 0,Y 263.346,Z 317.679,A -85,B 0,C 180,E1 -18164.522,E2 -18164.522} C_VEL
LIN {X 0,Y 263.369,Z 317.674,A -85,B 0,C 180,E1 -18169.234,E2 -18169.234} C_VEL
LIN {X 0,Y 263.568,Z 317.651,A -85,B 0,C 180,E1 -18172.339,E2 -18172.339} C_VEL
LIN {X 0,Y 263.746,Z 317.622,A -85,B 0,C 180,E1 -18178.473,E2 -18178.473} C_VEL
LIN {X 0,Y 263.745,Z 317.628,A -85,B 0,C 180,E1 -18181.527,E2 -18181.527} C_VEL
LIN {X 0,Y 263.528,Z 317.657,A -85,B 0,C 180,E1 -18187.663,E2 -18187.663} C_VEL
LIN {X 0,Y 263.35,Z 317.67,A -85,B 0,C 180,E1 -18190.767,E2 -18190.767} C_VEL
LIN {X 0,Y 263.346,Z 317.676,A -85,B 0,C 180,E1 -18195.479,E2 -18195.479} C_VEL
LIN {X 0,Y 263.258,Z 317.692,A -85,B 0,C 180,E1 -18200.308,E2 -18200.308} C_VEL
LIN {X 0,Y 263.164,Z 317.691,A -85,B 0,C 180,E1 -18205.296,E2 -18205.296} C_VEL
LIN {X 0,Y 263.132,Z 317.706,A -85,B 0,C 180,E1 -18208.736,E2 -18208.736} C_VEL
LIN {X 0,Y 263.125,Z 317.708,A -85,B 0,C 180,E1 -18212.29,E2 -18212.29} C_VEL
LIN {X 0,Y 263.178,Z 317.7,A -85,B 0,C 180,E1 -18216.764,E2 -18216.764} C_VEL
LIN {X 0,Y 263.122,Z 317.702,A -85,B 0,C 180,E1 -18221.595,E2 -18221.595} C_VEL
LIN {X 0,Y 263.1,Z 317.709,A -85,B 0,C 180,E1 -18226.013,E2 -18226.013} C_VEL
LIN {X 0,Y 263.09,Z 317.708,A -85,B 0,C 180,E1 -18230.126,E2 -18230.126} C_VEL
LIN {X 0,Y 263.161,Z 317.698,A -85,B 0,C 180,E1 -18234.019,E2 -18234.019} C_VEL
LIN {X 0,Y 263.128,Z 317.708,A -85,B 0,C 180,E1 -18237.712,E2 -18237.712} C_VEL
LIN {X 0,Y 263.148,Z 317.705,A -85,B 0,C 180,E1 -18241.806,E2 -18241.806} C_VEL
LIN {X 0,Y 263.19,Z 317.7,A -85,B 0,C 180,E1 -18245.219,E2 -18245.219} C_VEL
LIN {X 0,Y 263.24,Z 317.695,A -85,B 0,C 180,E1 -18249.693,E2 -18249.693} C_VEL
LIN {X 0,Y 263.317,Z 317.682,A -85,B 0,C 180,E1 -18254.521,E2 -18254.521} C_VEL
LIN {X 0,Y 263.355,Z 317.678,A -85,B 0,C 180,E1 -18259.235,E2 -18259.235} C_VEL
LIN {X 0,Y 263.529,Z 317.658,A -85,B 0,C 180,E1 -18262.338,E2 -18262.338} C_VEL
LIN {X 0,Y 263.728,Z 317.634,A -85,B 0,C 180,E1 -18268.474,E2 -18268.474} C_VEL
LIN {X 0,Y 263.728,Z 317.633,A -85,B 0,C 180,E1 -18271.528,E2 -18271.528} C_VEL
LIN {X 0,Y 263.519,Z 317.659,A -85,B 0,C 180,E1 -18277.664,E2 -18277.664} C_VEL
LIN {X 0,Y 263.33,Z 317.684,A -85,B 0,C 180,E1 -18280.768,E2 -18280.768} C_VEL
LIN {X 0,Y 263.292,Z 317.688,A -85,B 0,C 180,E1 -18285.482,E2 -18285.482} C_VEL
LIN {X 0,Y 263.223,Z 317.736,A -85,B 0,C 180,E1 -18288.385,E2 -18288.385} C_VEL
LIN {X 0,Y 263.367,Z 318.544,A -85,B 0,C 180,E1 -18288.627,E2 -18288.627} C_VEL
LIN {X 0,Y 272.098,Z 342.203,A -85,B 0,C 180,E1 -18290.161,E2 -18290.161} C_VEL
LIN {X 0,Y 275.541,Z 353.026,A -85,B 0,C 180,E1 -18290.788,E2 -18290.788} C_VEL
LIN {X 0,Y 272.802,Z 426.74,A -85,B 0,C 180,E1 -18292.984,E2 -18292.984} C_VEL
LIN {X 0,Y 271.887,Z 440.362,A -85,B 0,C 180,E1 -18293.696,E2 -18293.696} C_VEL
LIN {X 0,Y 270.917,Z 452.466,A -85,B 0,C 180,E1 -18294.622,E2 -18294.622} C_VEL
LIN {X 0,Y 269.551,Z 465.105,A -85,B 0,C 180,E1 -18295.92,E2 -18295.92} C_VEL
LIN {X 0,Y 268.27,Z 475.415,A -85,B 0,C 180,E1 -18297.271,E2 -18297.271} C_VEL
LIN {X 0,Y 266.893,Z 485.572,A -85,B 0,C 180,E1 -18298.92,E2 -18298.92} C_VEL
LIN {X 0,Y 265.487,Z 495.141,A -85,B 0,C 180,E1 -18300.858,E2 -18300.858} C_VEL
LIN {X 0,Y 264.099,Z 503.933,A -85,B 0,C 180,E1 -18303.062,E2 -18303.062} C_VEL
LIN {X 0,Y 263.11,Z 510.455,A -85,B 0,C 180,E1 -18305.086,E2 -18305.086} C_VEL
LIN {X 0,Y 262.303,Z 516.151,A -85,B 0,C 180,E1 -18307.265,E2 -18307.265} C_VEL
LIN {X 0,Y 261.761,Z 520.713,A -85,B 0,C 180,E1 -18309.467,E2 -18309.467} C_VEL
LIN {X 0,Y 261.121,Z 525.059,A -85,B 0,C 180,E1 -18312.29,E2 -18312.29} C_VEL
LIN {X 0,Y 260.86,Z 527.384,A -85,B 0,C 180,E1 -18314.467,E2 -18314.467} C_VEL
LIN {X 0,Y 260.807,Z 528.865,A -85,B 0,C 180,E1 -18316.684,E2 -18316.684} C_VEL
LIN {X 0,Y 260.999,Z 529.501,A -85,B 0,C 180,E1 -18319.739,E2 -18319.739} C_VEL
LIN {X 0,Y 261.308,Z 529.076,A -85,B 0,C 180,E1 -18321.786,E2 -18321.786} C_VEL
LIN {X 0,Y 261.823,Z 527.91,A -85,B 0,C 180,E1 -18323.804,E2 -18323.804} C_VEL
LIN {X 0,Y 262.919,Z 524.742,A -85,B 0,C 180,E1 -18326.903,E2 -18326.903} C_VEL
LIN {X 0,Y 264.307,Z 520.368,A -85,B 0,C 180,E1 -18329.654,E2 -18329.654} C_VEL
LIN {X 0,Y 265.922,Z 515.273,A -85,B 0,C 180,E1 -18332.023,E2 -18332.023} C_VEL
LIN {X 0,Y 267.946,Z 508.741,A -85,B 0,C 180,E1 -18334.376,E2 -18334.376} C_VEL
LIN {X 0,Y 270.365,Z 500.135,A -85,B 0,C 180,E1 -18336.788,E2 -18336.788} C_VEL
LIN {X 0,Y 272.836,Z 490.748,A -85,B 0,C 180,E1 -18338.861,E2 -18338.861} C_VEL
LIN {X 0,Y 275.235,Z 480.673,A -85,B 0,C 180,E1 -18340.612,E2 -18340.612} C_VEL
LIN {X 0,Y 277.486,Z 469.848,A -85,B 0,C 180,E1 -18342.115,E2 -18342.115} C_VEL
LIN {X 0,Y 279.473,Z 459.307,A -85,B 0,C 180,E1 -18343.265,E2 -18343.265} C_VEL
LIN {X 0,Y 281.203,Z 446.9,A -85,B 0,C 180,E1 -18344.322,E2 -18344.322} C_VEL
LIN {X 0,Y 282.514,Z 434.079,A -85,B 0,C 180,E1 -18345.112,E2 -18345.112} C_VEL
LIN {X 0,Y 283.516,Z 420.865,A -85,B 0,C 180,E1 -18345.622,E2 -18345.622} C_VEL
LIN {X 0,Y 286.748,Z 361.207,A -85,B 0,C 180,E1 -18347.383,E2 -18347.383} C_VEL
LIN {X 0,Y 281.74,Z 349.938,A -85,B 0,C 180,E1 -18348.671,E2 -18348.671} C_VEL
LIN {X 0,Y 280.053,Z 346.547,A -85,B 0,C 180,E1 -18349.113,E2 -18349.113} C_VEL
LIN {X 0,Y 277.367,Z 342.452,A -85,B 0,C 180,E1 -18349.783,E2 -18349.783} C_VEL
LIN {X 0,Y 274.128,Z 339.156,A -85,B 0,C 180,E1 -18350.552,E2 -18350.552} C_VEL
LIN {X 0,Y 265.03,Z 331.631,A -85,B 0,C 180,E1 -18352.855,E2 -18352.855} C_VEL
LIN {X 0,Y 263.032,Z 329.411,A -85,B 0,C 180,E1 -18353.435,E2 -18353.435} C_VEL
LIN {X 0,Y 260.182,Z 325.172,A -85,B 0,C 180,E1 -18354.366,E2 -18354.366} C_VEL
LIN {X 0,Y 256.945,Z 320.651,A -85,B 0,C 180,E1 -18355.489,E2 -18355.489} C_VEL
LIN {X 0,Y 256.481,Z 318.536,A -85,B 0,C 180,E1 -18356.661,E2 -18356.661} C_VEL
LIN {X 0,Y 256.761,Z 318.501,A -85,B 0,C 180,E1 -18360,E2 -18360} C_VEL
LIN {X 0,Y 256.497,Z 318.531,A -85,B 0,C 180,E1 -18363.141,E2 -18363.141} C_VEL
LIN {X 0,Y 256.498,Z 318.529,A -85,B 0,C 180,E1 -18367.874,E2 -18367.874} C_VEL
LIN {X 0,Y 256.292,Z 318.555,A -85,B 0,C 180,E1 -18372.672,E2 -18372.672} C_VEL
LIN {X 0,Y 256.236,Z 318.562,A -85,B 0,C 180,E1 -18376.264,E2 -18376.264} C_VEL
LIN {X 0,Y 256.144,Z 318.568,A -85,B 0,C 180,E1 -18381.11,E2 -18381.11} C_VEL
LIN {X 0,Y 256.173,Z 318.566,A -85,B 0,C 180,E1 -18385.129,E2 -18385.129} C_VEL
LIN {X 0,Y 256.113,Z 318.582,A -85,B 0,C 180,E1 -18389.6,E2 -18389.6} C_VEL
LIN {X 0,Y 256.07,Z 318.588,A -85,B 0,C 180,E1 -18393.292,E2 -18393.292} C_VEL
LIN {X 0,Y 256.116,Z 318.577,A -85,B 0,C 180,E1 -18397.27,E2 -18397.27} C_VEL
LIN {X 0,Y 256.056,Z 318.586,A -85,B 0,C 180,E1 -18401.203,E2 -18401.203} C_VEL
LIN {X 0,Y 256.042,Z 318.686,A -85,B 0,C 180,E1 -18405.307,E2 -18405.307} C_VEL
LIN {X 0,Y 258.076,Z 324.64,A -85,B 0,C 180,E1 -18408.671,E2 -18408.671} C_VEL
LIN {X 0,Y 259.912,Z 330.58,A -85,B 0,C 180,E1 -18411.643,E2 -18411.643} C_VEL
LIN {X 0,Y 260.552,Z 332.667,A -85,B 0,C 180,E1 -18412.555,E2 -18412.555} C_VEL
LIN {X 0,Y 264.434,Z 339.438,A -85,B 0,C 180,E1 -18413.825,E2 -18413.825} C_VEL
LIN {X 0,Y 269.429,Z 348.504,A -85,B 0,C 180,E1 -18415.349,E2 -18415.349} C_VEL
LIN {X 0,Y 275.275,Z 360.884,A -85,B 0,C 180,E1 -18417.049,E2 -18417.049} C_VEL
LIN {X 0,Y 276.936,Z 365.346,A -85,B 0,C 180,E1 -18417.543,E2 -18417.543} C_VEL
LIN {X 0,Y 279.314,Z 381.609,A -85,B 0,C 180,E1 -18418.635,E2 -18418.635} C_VEL
LIN {X 0,Y 280.03,Z 388.186,A -85,B 0,C 180,E1 -18419.013,E2 -18419.013} C_VEL
LIN {X 0,Y 276.779,Z 444.07,A -85,B 0,C 180,E1 -18420.722,E2 -18420.722} C_VEL
LIN {X 0,Y 275.333,Z 457.672,A -85,B 0,C 180,E1 -18421.405,E2 -18421.405} C_VEL
LIN {X 0,Y 273.478,Z 469.493,A -85,B 0,C 180,E1 -18422.238,E2 -18422.238} C_VEL
LIN {X 0,Y 271.175,Z 481.884,A -85,B 0,C 180,E1 -18423.444,E2 -18423.444} C_VEL
LIN {X 0,Y 268.574,Z 493.08,A -85,B 0,C 180,E1 -18424.834,E2 -18424.834} C_VEL
LIN {X 0,Y 266.107,Z 503.263,A -85,B 0,C 180,E1 -18426.455,E2 -18426.455} C_VEL
LIN {X 0,Y 263.379,Z 513.363,A -85,B 0,C 180,E1 -18428.474,E2 -18428.474} C_VEL
LIN {X 0,Y 261.125,Z 521.106,A -85,B 0,C 180,E1 -18430.39,E2 -18430.39} C_VEL
LIN {X 0,Y 259.077,Z 528.41,A -85,B 0,C 180,E1 -18432.638,E2 -18432.638} C_VEL
LIN {X 0,Y 257.24,Z 534.453,A -85,B 0,C 180,E1 -18434.956,E2 -18434.956} C_VEL
LIN {X 0,Y 255.777,Z 539.257,A -85,B 0,C 180,E1 -18437.301,E2 -18437.301} C_VEL
LIN {X 0,Y 254.895,Z 542.958,A -85,B 0,C 180,E1 -18439.675,E2 -18439.675} C_VEL
LIN {X 0,Y 254.306,Z 545.664,A -85,B 0,C 180,E1 -18442.057,E2 -18442.057} C_VEL
LIN {X 0,Y 253.99,Z 547.705,A -85,B 0,C 180,E1 -18444.96,E2 -18444.96} C_VEL
LIN {X 0,Y 254.018,Z 548.257,A -85,B 0,C 180,E1 -18446.827,E2 -18446.827} C_VEL
LIN {X 0,Y 254.071,Z 548.307,A -85,B 0,C 180,E1 -18448.414,E2 -18448.414} C_VEL
LIN {X 0,Y 254.102,Z 547.954,A -85,B 0,C 180,E1 -18449.999,E2 -18449.999} C_VEL
LIN {X 0,Y 254.086,Z 547.143,A -85,B 0,C 180,E1 -18451.584,E2 -18451.584} C_VEL
LIN {X 0,Y 254.069,Z 545.903,A -85,B 0,C 180,E1 -18453.17,E2 -18453.17} C_VEL
LIN {X 0,Y 254.084,Z 543.592,A -85,B 0,C 180,E1 -18455.276,E2 -18455.276} C_VEL
LIN {X 0,Y 254.311,Z 539.445,A -85,B 0,C 180,E1 -18457.941,E2 -18457.941} C_VEL
LIN {X 0,Y 254.748,Z 534.494,A -85,B 0,C 180,E1 -18460.329,E2 -18460.329} C_VEL
LIN {X 0,Y 255.51,Z 528.216,A -85,B 0,C 180,E1 -18462.711,E2 -18462.711} C_VEL
LIN {X 0,Y 256.712,Z 520.369,A -85,B 0,C 180,E1 -18465.074,E2 -18465.074} C_VEL
LIN {X 0,Y 257.961,Z 512.3,A -85,B 0,C 180,E1 -18467.029,E2 -18467.029} C_VEL
LIN {X 0,Y 259.43,Z 502.443,A -85,B 0,C 180,E1 -18468.969,E2 -18468.969} C_VEL
LIN {X 0,Y 261.016,Z 491.509,A -85,B 0,C 180,E1 -18470.694,E2 -18470.694} C_VEL
LIN {X 0,Y 262.429,Z 480.863,A -85,B 0,C 180,E1 -18472.019,E2 -18472.019} C_VEL
LIN {X 0,Y 263.832,Z 469.321,A -85,B 0,C 180,E1 -18473.135,E2 -18473.135} C_VEL
LIN {X 0,Y 265.143,Z 455.765,A -85,B 0,C 180,E1 -18474.101,E2 -18474.101} C_VEL
LIN {X 0,Y 265.943,Z 443.015,A -85,B 0,C 180,E1 -18474.699,E2 -18474.699} C_VEL
LIN {X 0,Y 267.935,Z 384.279,A -85,B 0,C 180,E1 -18476.496,E2 -18476.496} C_VEL
LIN {X 0,Y 262.806,Z 345.354,A -85,B 0,C 180,E1 -18478.22,E2 -18478.22} C_VEL
LIN {X 0,Y 259.932,Z 336.614,A -85,B 0,C 180,E1 -18478.805,E2 -18478.805} C_VEL
LIN {X 0,Y 257.44,Z 324.693,A -85,B 0,C 180,E1 -18483.091,E2 -18483.091} C_VEL
LIN {X 0,Y 256.168,Z 318.58,A -85,B 0,C 180,E1 -18485.419,E2 -18485.419} C_VEL
LIN {X 0,Y 256.057,Z 318.591,A -85,B 0,C 180,E1 -18489.779,E2 -18489.779} C_VEL
LIN {X 0,Y 256.045,Z 318.589,A -85,B 0,C 180,E1 -18493.329,E2 -18493.329} C_VEL
LIN {X 0,Y 256.066,Z 318.587,A -85,B 0,C 180,E1 -18497.819,E2 -18497.819} C_VEL
LIN {X 0,Y 256.084,Z 318.587,A -85,B 0,C 180,E1 -18500.86,E2 -18500.86} C_VEL
LIN {X 0,Y 256.116,Z 318.583,A -85,B 0,C 180,E1 -18504.813,E2 -18504.813} C_VEL
LIN {X 0,Y 256.087,Z 318.579,A -85,B 0,C 180,E1 -18508.572,E2 -18508.572} C_VEL
LIN {X 0,Y 256.136,Z 318.574,A -85,B 0,C 180,E1 -18512.196,E2 -18512.196} C_VEL
LIN {X 0,Y 256.162,Z 318.576,A -85,B 0,C 180,E1 -18515.699,E2 -18515.699} C_VEL
LIN {X 0,Y 256.162,Z 318.575,A -85,B 0,C 180,E1 -18519.105,E2 -18519.105} C_VEL
LIN {X 0,Y 256.295,Z 318.558,A -85,B 0,C 180,E1 -18524.085,E2 -18524.085} C_VEL
LIN {X 0,Y 256.305,Z 318.552,A -85,B 0,C 180,E1 -18528.934,E2 -18528.934} C_VEL
LIN {X 0,Y 256.535,Z 318.528,A -85,B 0,C 180,E1 -18532.127,E2 -18532.127} C_VEL
LIN {X 0,Y 256.709,Z 318.498,A -85,B 0,C 180,E1 -18538.432,E2 -18538.432} C_VEL
LIN {X 0,Y 256.708,Z 318.504,A -85,B 0,C 180,E1 -18541.569,E2 -18541.569} C_VEL
LIN {X 0,Y 256.451,Z 318.536,A -85,B 0,C 180,E1 -18546.569,E2 -18546.569} C_VEL
LIN {X 0,Y 256.422,Z 318.537,A -85,B 0,C 180,E1 -18549.466,E2 -18549.466} C_VEL
LIN {X 0,Y 256.251,Z 318.562,A -85,B 0,C 180,E1 -18554.291,E2 -18554.291} C_VEL
LIN {X 0,Y 256.206,Z 318.567,A -85,B 0,C 180,E1 -18557.563,E2 -18557.563} C_VEL
LIN {X 0,Y 256.148,Z 318.572,A -85,B 0,C 180,E1 -18561.118,E2 -18561.118} C_VEL
LIN {X 0,Y 256.129,Z 318.567,A -85,B 0,C 180,E1 -18565.113,E2 -18565.113} C_VEL
LIN {X 0,Y 256.052,Z 318.585,A -85,B 0,C 180,E1 -18569.608,E2 -18569.608} C_VEL
LIN {X 0,Y 256.063,Z 318.586,A -85,B 0,C 180,E1 -18573.294,E2 -18573.294} C_VEL
LIN {X 0,Y 256.11,Z 318.576,A -85,B 0,C 180,E1 -18577.271,E2 -18577.271} C_VEL
LIN {X 0,Y 256.052,Z 318.584,A -85,B 0,C 180,E1 -18581.205,E2 -18581.205} C_VEL
LIN {X 0,Y 256.038,Z 318.59,A -85,B 0,C 180,E1 -18585.536,E2 -18585.536} C_VEL
LIN {X 0,Y 256.039,Z 318.591,A -85,B 0,C 180,E1 -18588.795,E2 -18588.795} C_VEL
LIN {X 0,Y 256.128,Z 318.574,A -85,B 0,C 180,E1 -18592.868,E2 -18592.868} C_VEL
LIN {X 0,Y 256.066,Z 318.586,A -85,B 0,C 180,E1 -18596.708,E2 -18596.708} C_VEL
LIN {X 0,Y 256.055,Z 318.586,A -85,B 0,C 180,E1 -18600.394,E2 -18600.394} C_VEL
LIN {X 0,Y 256.134,Z 318.578,A -85,B 0,C 180,E1 -18604.89,E2 -18604.89} C_VEL
LIN {X 0,Y 256.149,Z 318.576,A -85,B 0,C 180,E1 -18609.105,E2 -18609.105} C_VEL
LIN {X 0,Y 256.251,Z 318.564,A -85,B 0,C 180,E1 -18614.083,E2 -18614.083} C_VEL
LIN {X 0,Y 256.291,Z 318.558,A -85,B 0,C 180,E1 -18617.329,E2 -18617.329} C_VEL
LIN {X 0,Y 256.437,Z 318.539,A -85,B 0,C 180,E1 -18620.624,E2 -18620.624} C_VEL
LIN {X 0,Y 256.456,Z 318.54,A -85,B 0,C 180,E1 -18623.708,E2 -18623.708} C_VEL
LIN {X 0,Y 256.689,Z 318.512,A -85,B 0,C 180,E1 -18628.432,E2 -18628.432} C_VEL
LIN {X 0,Y 256.689,Z 318.51,A -85,B 0,C 180,E1 -18631.57,E2 -18631.57} C_VEL
LIN {X 0,Y 256.453,Z 318.542,A -85,B 0,C 180,E1 -18636.294,E2 -18636.294} C_VEL
LIN {X 0,Y 256.403,Z 318.545,A -85,B 0,C 180,E1 -18639.467,E2 -18639.467} C_VEL
LIN {X 0,Y 256.199,Z 318.573,A -85,B 0,C 180,E1 -18644.294,E2 -18644.294} C_VEL
LIN {X 0,Y 256.17,Z 318.639,A -85,B 0,C 180,E1 -18647.978,E2 -18647.978} C_VEL
LIN {X 0,Y 258.185,Z 323.991,A -85,B 0,C 180,E1 -18648.35,E2 -18648.35} C_VEL
LIN {X 0,Y 266.872,Z 347.814,A -85,B 0,C 180,E1 -18649.921,E2 -18649.921} C_VEL
LIN {X 0,Y 268.825,Z 354.302,A -85,B 0,C 180,E1 -18650.293,E2 -18650.293} C_VEL
LIN {X 0,Y 266.063,Z 426.847,A -85,B 0,C 180,E1 -18652.516,E2 -18652.516} C_VEL
LIN {X 0,Y 265.115,Z 440.687,A -85,B 0,C 180,E1 -18653.258,E2 -18653.258} C_VEL
LIN {X 0,Y 264.036,Z 453.355,A -85,B 0,C 180,E1 -18654.263,E2 -18654.263} C_VEL
LIN {X 0,Y 262.677,Z 465.573,A -85,B 0,C 180,E1 -18655.559,E2 -18655.559} C_VEL
LIN {X 0,Y 261.304,Z 476.18,A -85,B 0,C 180,E1 -18656.993,E2 -18656.993} C_VEL
LIN {X 0,Y 259.911,Z 486.207,A -85,B 0,C 180,E1 -18658.683,E2 -18658.683} C_VEL
LIN {X 0,Y 258.341,Z 496.191,A -85,B 0,C 180,E1 -18660.781,E2 -18660.781} C_VEL
LIN {X 0,Y 257.21,Z 503.364,A -85,B 0,C 180,E1 -18662.629,E2 -18662.629} C_VEL
LIN {X 0,Y 256.213,Z 509.781,A -85,B 0,C 180,E1 -18664.622,E2 -18664.622} C_VEL
LIN {X 0,Y 255.21,Z 516.668,A -85,B 0,C 180,E1 -18667.29,E2 -18667.29} C_VEL
LIN {X 0,Y 254.691,Z 520.915,A -85,B 0,C 180,E1 -18669.408,E2 -18669.408} C_VEL
LIN {X 0,Y 254.144,Z 524.499,A -85,B 0,C 180,E1 -18671.698,E2 -18671.698} C_VEL
LIN {X 0,Y 253.812,Z 527.072,A -85,B 0,C 180,E1 -18673.95,E2 -18673.95} C_VEL
LIN {X 0,Y 253.72,Z 528.762,A -85,B 0,C 180,E1 -18676.171,E2 -18676.171} C_VEL
LIN {X 0,Y 253.81,Z 529.655,A -85,B 0,C 180,E1 -18678.386,E2 -18678.386} C_VEL
LIN {X 0,Y 254.034,Z 529.723,A -85,B 0,C 180,E1 -18680.773,E2 -18680.773} C_VEL
LIN {X 0,Y 254.553,Z 528.836,A -85,B 0,C 180,E1 -18683.195,E2 -18683.195} C_VEL
LIN {X 0,Y 255.307,Z 526.939,A -85,B 0,C 180,E1 -18685.674,E2 -18685.674} C_VEL
LIN {X 0,Y 256.639,Z 523.239,A -85,B 0,C 180,E1 -18688.646,E2 -18688.646} C_VEL
LIN {X 0,Y 257.881,Z 519.707,A -85,B 0,C 180,E1 -18690.704,E2 -18690.704} C_VEL
LIN {X 0,Y 259.77,Z 514.044,A -85,B 0,C 180,E1 -18693.229,E2 -18693.229} C_VEL
LIN {X 0,Y 262.111,Z 506.762,A -85,B 0,C 180,E1 -18695.735,E2 -18695.735} C_VEL
LIN {X 0,Y 264.261,Z 499.475,A -85,B 0,C 180,E1 -18697.729,E2 -18697.729} C_VEL
LIN {X 0,Y 266.82,Z 490.157,A -85,B 0,C 180,E1 -18699.774,E2 -18699.774} C_VEL
LIN {X 0,Y 269.48,Z 479.642,A -85,B 0,C 180,E1 -18701.6,E2 -18701.6} C_VEL
LIN {X 0,Y 271.813,Z 468.965,A -85,B 0,C 180,E1 -18703.074,E2 -18703.074} C_VEL
LIN {X 0,Y 273.882,Z 457.808,A -85,B 0,C 180,E1 -18704.273,E2 -18704.273} C_VEL
LIN {X 0,Y 275.691,Z 444.832,A -85,B 0,C 180,E1 -18705.346,E2 -18705.346} C_VEL
LIN {X 0,Y 277.07,Z 431.907,A -85,B 0,C 180,E1 -18706.088,E2 -18706.088} C_VEL
LIN {X 0,Y 278.147,Z 415.689,A -85,B 0,C 180,E1 -18706.654,E2 -18706.654} C_VEL
LIN {X 0,Y 281.102,Z 363.248,A -85,B 0,C 180,E1 -18708.243,E2 -18708.243} C_VEL
LIN {X 0,Y 275.43,Z 350.803,A -85,B 0,C 180,E1 -18709.793,E2 -18709.793} C_VEL
LIN {X 0,Y 270.08,Z 340.978,A -85,B 0,C 180,E1 -18711.3,E2 -18711.3} C_VEL
LIN {X 0,Y 263.635,Z 330.123,A -85,B 0,C 180,E1 -18713.254,E2 -18713.254} C_VEL
LIN {X 0,Y 263.032,Z 329.411,A -85,B 0,C 180,E1 -18713.435,E2 -18713.435} C_VEL
LIN {X 0,Y 260.925,Z 327.576,A -85,B 0,C 180,E1 -18714.054,E2 -18714.054} C_VEL
LIN {X 0,Y 252.919,Z 324.604,A -85,B 0,C 180,E1 -18716.379,E2 -18716.379} C_VEL
LIN {X 0,Y 250.933,Z 322.884,A -85,B 0,C 180,E1 -18717.065,E2 -18717.065} C_VEL
LIN {X 0,Y 249.995,Z 321.201,A -85,B 0,C 180,E1 -18717.482,E2 -18717.482} C_VEL
LIN {X 0,Y 249.669,Z 319.381,A -85,B 0,C 180,E1 -18718.588,E2 -18718.588} C_VEL
LIN {X 0,Y 249.677,Z 319.379,A -85,B 0,C 180,E1 -18721.613,E2 -18721.613} C_VEL
LIN {X 0,Y 249.44,Z 319.406,A -85,B 0,C 180,E1 -18726.471,E2 -18726.471} C_VEL
LIN {X 0,Y 249.346,Z 319.417,A -85,B 0,C 180,E1 -18729.736,E2 -18729.736} C_VEL
LIN {X 0,Y 249.181,Z 319.441,A -85,B 0,C 180,E1 -18734.705,E2 -18734.705} C_VEL
LIN {X 0,Y 249.115,Z 319.447,A -85,B 0,C 180,E1 -18738.079,E2 -18738.079} C_VEL
LIN {X 0,Y 249.083,Z 319.449,A -85,B 0,C 180,E1 -18741.518,E2 -18741.518} C_VEL
LIN {X 0,Y 249.12,Z 319.446,A -85,B 0,C 180,E1 -18745.475,E2 -18745.475} C_VEL
LIN {X 0,Y 249.082,Z 319.451,A -85,B 0,C 180,E1 -18748.991,E2 -18748.991} C_VEL
LIN {X 0,Y 249.033,Z 319.459,A -85,B 0,C 180,E1 -18752.425,E2 -18752.425} C_VEL
LIN {X 0,Y 249.05,Z 319.464,A -85,B 0,C 180,E1 -18756.342,E2 -18756.342} C_VEL
LIN {X 0,Y 249.008,Z 319.463,A -85,B 0,C 180,E1 -18760.478,E2 -18760.478} C_VEL
LIN {X 0,Y 249.026,Z 319.546,A -85,B 0,C 180,E1 -18763.339,E2 -18763.339} C_VEL
LIN {X 0,Y 251.189,Z 325.882,A -85,B 0,C 180,E1 -18767.275,E2 -18767.275} C_VEL
LIN {X 0,Y 253.197,Z 332.081,A -85,B 0,C 180,E1 -18770.568,E2 -18770.568} C_VEL
LIN {X 0,Y 256.133,Z 336.997,A -85,B 0,C 180,E1 -18771.642,E2 -18771.642} C_VEL
LIN {X 0,Y 260.329,Z 344.161,A -85,B 0,C 180,E1 -18773.088,E2 -18773.088} C_VEL
LIN {X 0,Y 265.329,Z 353.534,A -85,B 0,C 180,E1 -18774.698,E2 -18774.698} C_VEL
LIN {X 0,Y 270.783,Z 365.434,A -85,B 0,C 180,E1 -18776.384,E2 -18776.384} C_VEL
LIN {X 0,Y 271.885,Z 368.411,A -85,B 0,C 180,E1 -18776.726,E2 -18776.726} C_VEL
LIN {X 0,Y 274.047,Z 384.457,A -85,B 0,C 180,E1 -18777.81,E2 -18777.81} C_VEL
LIN {X 0,Y 274.454,Z 390.649,A -85,B 0,C 180,E1 -18778.143,E2 -18778.143} C_VEL
LIN {X 0,Y 271.12,Z 444.336,A -85,B 0,C 180,E1 -18779.836,E2 -18779.836} C_VEL
LIN {X 0,Y 269.602,Z 457.724,A -85,B 0,C 180,E1 -18780.525,E2 -18780.525} C_VEL
LIN {X 0,Y 267.672,Z 469.451,A -85,B 0,C 180,E1 -18781.368,E2 -18781.368} C_VEL
LIN {X 0,Y 265.264,Z 481.782,A -85,B 0,C 180,E1 -18782.59,E2 -18782.59} C_VEL
LIN {X 0,Y 262.515,Z 492.957,A -85,B 0,C 180,E1 -18783.998,E2 -18783.998} C_VEL
LIN {X 0,Y 259.995,Z 503.104,A -85,B 0,C 180,E1 -18785.654,E2 -18785.654} C_VEL
LIN {X 0,Y 257.339,Z 512.324,A -85,B 0,C 180,E1 -18787.52,E2 -18787.52} C_VEL
LIN {X 0,Y 254.872,Z 520.269,A -85,B 0,C 180,E1 -18789.502,E2 -18789.502} C_VEL
LIN {X 0,Y 252.698,Z 527.558,A -85,B 0,C 180,E1 -18791.766,E2 -18791.766} C_VEL
LIN {X 0,Y 250.395,Z 534.635,A -85,B 0,C 180,E1 -18794.535,E2 -18794.535} C_VEL
LIN {X 0,Y 248.823,Z 539.343,A -85,B 0,C 180,E1 -18796.94,E2 -18796.94} C_VEL
LIN {X 0,Y 247.876,Z 542.958,A -85,B 0,C 180,E1 -18799.379,E2 -18799.379} C_VEL
LIN {X 0,Y 247.257,Z 545.57,A -85,B 0,C 180,E1 -18801.829,E2 -18801.829} C_VEL
LIN {X 0,Y 247.007,Z 546.797,A -85,B 0,C 180,E1 -18803.464,E2 -18803.464} C_VEL
LIN {X 0,Y 246.902,Z 547.596,A -85,B 0,C 180,E1 -18805.1,E2 -18805.1} C_VEL
LIN {X 0,Y 246.914,Z 548.005,A -85,B 0,C 180,E1 -18806.736,E2 -18806.736} C_VEL
LIN {X 0,Y 246.999,Z 548.018,A -85,B 0,C 180,E1 -18808.369,E2 -18808.369} C_VEL
LIN {X 0,Y 247.029,Z 547.605,A -85,B 0,C 180,E1 -18809.999,E2 -18809.999} C_VEL
LIN {X 0,Y 247.015,Z 546.74,A -85,B 0,C 180,E1 -18811.629,E2 -18811.629} C_VEL
LIN {X 0,Y 246.986,Z 545.459,A -85,B 0,C 180,E1 -18813.261,E2 -18813.261} C_VEL
LIN {X 0,Y 246.986,Z 543.399,A -85,B 0,C 180,E1 -18815.174,E2 -18815.174} C_VEL
LIN {X 0,Y 247.258,Z 538.827,A -85,B 0,C 180,E1 -18818.169,E2 -18818.169} C_VEL
LIN {X 0,Y 247.736,Z 533.779,A -85,B 0,C 180,E1 -18820.625,E2 -18820.625} C_VEL
LIN {X 0,Y 248.539,Z 527.39,A -85,B 0,C 180,E1 -18823.073,E2 -18823.073} C_VEL
LIN {X 0,Y 249.778,Z 519.353,A -85,B 0,C 180,E1 -18825.503,E2 -18825.503} C_VEL
LIN {X 0,Y 251.068,Z 511.13,A -85,B 0,C 180,E1 -18827.512,E2 -18827.512} C_VEL
LIN {X 0,Y 252.674,Z 501.104,A -85,B 0,C 180,E1 -18829.497,E2 -18829.497} C_VEL
LIN {X 0,Y 254.136,Z 491.255,A -85,B 0,C 180,E1 -18831.069,E2 -18831.069} C_VEL
LIN {X 0,Y 255.585,Z 480.607,A -85,B 0,C 180,E1 -18832.427,E2 -18832.427} C_VEL
LIN {X 0,Y 257.02,Z 469.066,A -85,B 0,C 180,E1 -18833.571,E2 -18833.571} C_VEL
LIN {X 0,Y 258.37,Z 455.525,A -85,B 0,C 180,E1 -18834.56,E2 -18834.56} C_VEL
LIN {X 0,Y 259.201,Z 442.815,A -85,B 0,C 180,E1 -18835.172,E2 -18835.172} C_VEL
LIN {X 0,Y 261.248,Z 385.028,A -85,B 0,C 180,E1 -18836.989,E2 -18836.989} C_VEL
LIN {X 0,Y 256.232,Z 347.074,A -85,B 0,C 180,E1 -18838.733,E2 -18838.733} C_VEL
LIN {X 0,Y 252.644,Z 336.389,A -85,B 0,C 180,E1 -18839.472,E2 -18839.472} C_VEL
